(* IEC 61131-3 sources: LTL-Test-Case-Generation/ (part 3) *)

(* ---- SF_ModeSelector_Test.st ---- *)
FUNCTION_BLOCK SF_ModeSelector_Test
VAR_INPUT
END_VAR
VAR_OUTPUT
	failed_0: BOOL := FALSE;
	finished_0: BOOL := FALSE;
END_VAR
VAR
	fb_0: SF_ModeSelector_BranchCounters;
	waitCounter_0: UINT := 0;
	testState_0: UINT := 0;
END_VAR

IF NOT failed_0 AND NOT finished_0 THEN
CASE testState_0 OF
0:
	fb_0.Activate := FALSE;
	fb_0();
	failed_0 := NOT (((((((((((((((((NOT (fb_0.Reset_Before) AND NOT (fb_0.S_SetMode_Before)) AND NOT (fb_0.T_1.Q)) AND (fb_0.DiagCode = 0)) AND NOT (fb_0.Ready)) AND NOT (fb_0.SafetyDemand)) AND NOT (fb_0.ResetRequest)) AND NOT (fb_0.Error)) AND NOT (fb_0.S_AnyModeSel)) AND NOT (fb_0.S_Mode0Sel)) AND NOT (fb_0.S_Mode1Sel)) AND NOT (fb_0.S_Mode2Sel)) AND NOT (fb_0.S_Mode3Sel)) AND NOT (fb_0.S_Mode4Sel)) AND NOT (fb_0.S_Mode5Sel)) AND NOT (fb_0.S_Mode6Sel)) AND NOT (fb_0.S_Mode7Sel)));
	testState_0 := testState_0 + 1;
1:
	fb_0.Activate := TRUE; fb_0.AutoSetMode := TRUE; fb_0.S_SetMode := FALSE; fb_0.S_Unlock := FALSE; fb_0.Reset := FALSE; fb_0.S_Mode0 := FALSE; fb_0.S_Mode1 := FALSE; fb_0.S_Mode2 := FALSE; fb_0.S_Mode3 := FALSE; fb_0.S_Mode4 := FALSE; fb_0.S_Mode5 := FALSE; fb_0.S_Mode6 := FALSE; fb_0.S_Mode7 := FALSE;
	fb_0();
	failed_0 := NOT (((((((((((((((((NOT (fb_0.Reset_Before) AND NOT (fb_0.S_SetMode_Before)) AND NOT (fb_0.T_1.Q)) AND (fb_0.DiagCode = 34818)) AND fb_0.Ready) AND fb_0.SafetyDemand) AND NOT (fb_0.ResetRequest)) AND NOT (fb_0.Error)) AND NOT (fb_0.S_AnyModeSel)) AND NOT (fb_0.S_Mode0Sel)) AND NOT (fb_0.S_Mode1Sel)) AND NOT (fb_0.S_Mode2Sel)) AND NOT (fb_0.S_Mode3Sel)) AND NOT (fb_0.S_Mode4Sel)) AND NOT (fb_0.S_Mode5Sel)) AND NOT (fb_0.S_Mode6Sel)) AND NOT (fb_0.S_Mode7Sel)));
	testState_0 := testState_0 + 1;
2:
	IF fb_0.T_1.Q THEN
		waitCounter_0 := 0;
		testState_0 := testState_0 + 1;
	ELSE
		failed_0 := NOT ((NOT (fb_0.Reset_Before) AND (NOT (fb_0.S_SetMode_Before) AND (NOT (fb_0.T_1.Q) AND ((fb_0.DiagCode = 34818) AND (fb_0.Ready AND (fb_0.SafetyDemand AND (NOT (fb_0.ResetRequest) AND (NOT (fb_0.Error) AND (NOT (fb_0.S_AnyModeSel) AND (NOT (fb_0.S_Mode0Sel) AND (NOT (fb_0.S_Mode1Sel) AND (NOT (fb_0.S_Mode2Sel) AND (NOT (fb_0.S_Mode3Sel) AND (NOT (fb_0.S_Mode4Sel) AND (NOT (fb_0.S_Mode5Sel) AND (NOT (fb_0.S_Mode6Sel) AND NOT (fb_0.S_Mode7Sel))))))))))))))))));
		IF waitCounter_0 > 100 THEN
			finished_0 := TRUE;
		ELSE
			waitCounter_0 := waitCounter_0 + 1;
			fb_0();
		END_IF
	END_IF
3:
	failed_0 := NOT (((((((((((((((((NOT (fb_0.Reset_Before) AND NOT (fb_0.S_SetMode_Before)) AND fb_0.T_1.Q) AND (fb_0.DiagCode = 49184)) AND fb_0.Ready) AND NOT (fb_0.SafetyDemand)) AND NOT (fb_0.ResetRequest)) AND fb_0.Error) AND NOT (fb_0.S_AnyModeSel)) AND NOT (fb_0.S_Mode0Sel)) AND NOT (fb_0.S_Mode1Sel)) AND NOT (fb_0.S_Mode2Sel)) AND NOT (fb_0.S_Mode3Sel)) AND NOT (fb_0.S_Mode4Sel)) AND NOT (fb_0.S_Mode5Sel)) AND NOT (fb_0.S_Mode6Sel)) AND NOT (fb_0.S_Mode7Sel)));
	testState_0 := testState_0 + 1;
4:
	fb_0.Activate := TRUE; fb_0.AutoSetMode := TRUE; fb_0.S_SetMode := FALSE; fb_0.S_Unlock := FALSE; fb_0.Reset := TRUE; fb_0.S_Mode0 := FALSE; fb_0.S_Mode1 := FALSE; fb_0.S_Mode2 := FALSE; fb_0.S_Mode3 := FALSE; fb_0.S_Mode4 := FALSE; fb_0.S_Mode5 := FALSE; fb_0.S_Mode6 := FALSE; fb_0.S_Mode7 := FALSE;
	fb_0();
	failed_0 := NOT (((((((((((((((((fb_0.Reset_Before AND NOT (fb_0.S_SetMode_Before)) AND fb_0.T_1.Q) AND (fb_0.DiagCode = 49184)) AND fb_0.Ready) AND NOT (fb_0.SafetyDemand)) AND NOT (fb_0.ResetRequest)) AND fb_0.Error) AND NOT (fb_0.S_AnyModeSel)) AND NOT (fb_0.S_Mode0Sel)) AND NOT (fb_0.S_Mode1Sel)) AND NOT (fb_0.S_Mode2Sel)) AND NOT (fb_0.S_Mode3Sel)) AND NOT (fb_0.S_Mode4Sel)) AND NOT (fb_0.S_Mode5Sel)) AND NOT (fb_0.S_Mode6Sel)) AND NOT (fb_0.S_Mode7Sel)));
	testState_0 := testState_0 + 1;
5:
	fb_0.Activate := TRUE; fb_0.AutoSetMode := TRUE; fb_0.S_SetMode := FALSE; fb_0.S_Unlock := FALSE; fb_0.Reset := TRUE; fb_0.S_Mode0 := FALSE; fb_0.S_Mode1 := FALSE; fb_0.S_Mode2 := FALSE; fb_0.S_Mode3 := FALSE; fb_0.S_Mode4 := FALSE; fb_0.S_Mode5 := FALSE; fb_0.S_Mode6 := FALSE; fb_0.S_Mode7 := FALSE;
	fb_0();
	failed_0 := NOT (((((((((((((((((fb_0.Reset_Before AND NOT (fb_0.S_SetMode_Before)) AND fb_0.T_1.Q) AND (fb_0.DiagCode = 49185)) AND fb_0.Ready) AND NOT (fb_0.SafetyDemand)) AND NOT (fb_0.ResetRequest)) AND fb_0.Error) AND NOT (fb_0.S_AnyModeSel)) AND NOT (fb_0.S_Mode0Sel)) AND NOT (fb_0.S_Mode1Sel)) AND NOT (fb_0.S_Mode2Sel)) AND NOT (fb_0.S_Mode3Sel)) AND NOT (fb_0.S_Mode4Sel)) AND NOT (fb_0.S_Mode5Sel)) AND NOT (fb_0.S_Mode6Sel)) AND NOT (fb_0.S_Mode7Sel)));
	testState_0 := testState_0 + 1;
6:
	fb_0.Activate := TRUE; fb_0.AutoSetMode := TRUE; fb_0.S_SetMode := FALSE; fb_0.S_Unlock := FALSE; fb_0.Reset := TRUE; fb_0.S_Mode0 := FALSE; fb_0.S_Mode1 := FALSE; fb_0.S_Mode2 := FALSE; fb_0.S_Mode3 := FALSE; fb_0.S_Mode4 := FALSE; fb_0.S_Mode5 := FALSE; fb_0.S_Mode6 := FALSE; fb_0.S_Mode7 := FALSE;
	fb_0();
	failed_0 := NOT (((((((((((((((((fb_0.Reset_Before AND NOT (fb_0.S_SetMode_Before)) AND fb_0.T_1.Q) AND (fb_0.DiagCode = 49185)) AND fb_0.Ready) AND NOT (fb_0.SafetyDemand)) AND NOT (fb_0.ResetRequest)) AND fb_0.Error) AND NOT (fb_0.S_AnyModeSel)) AND NOT (fb_0.S_Mode0Sel)) AND NOT (fb_0.S_Mode1Sel)) AND NOT (fb_0.S_Mode2Sel)) AND NOT (fb_0.S_Mode3Sel)) AND NOT (fb_0.S_Mode4Sel)) AND NOT (fb_0.S_Mode5Sel)) AND NOT (fb_0.S_Mode6Sel)) AND NOT (fb_0.S_Mode7Sel)));
	testState_0 := testState_0 + 1;
7:
	fb_0.Activate := TRUE; fb_0.AutoSetMode := TRUE; fb_0.S_SetMode := FALSE; fb_0.S_Unlock := FALSE; fb_0.Reset := FALSE; fb_0.S_Mode0 := FALSE; fb_0.S_Mode1 := FALSE; fb_0.S_Mode2 := FALSE; fb_0.S_Mode3 := FALSE; fb_0.S_Mode4 := FALSE; fb_0.S_Mode5 := FALSE; fb_0.S_Mode6 := FALSE; fb_0.S_Mode7 := FALSE;
	fb_0();
	failed_0 := NOT (((((((((((((((((NOT (fb_0.Reset_Before) AND NOT (fb_0.S_SetMode_Before)) AND fb_0.T_1.Q) AND (fb_0.DiagCode = 49184)) AND fb_0.Ready) AND NOT (fb_0.SafetyDemand)) AND NOT (fb_0.ResetRequest)) AND fb_0.Error) AND NOT (fb_0.S_AnyModeSel)) AND NOT (fb_0.S_Mode0Sel)) AND NOT (fb_0.S_Mode1Sel)) AND NOT (fb_0.S_Mode2Sel)) AND NOT (fb_0.S_Mode3Sel)) AND NOT (fb_0.S_Mode4Sel)) AND NOT (fb_0.S_Mode5Sel)) AND NOT (fb_0.S_Mode6Sel)) AND NOT (fb_0.S_Mode7Sel)));
	testState_0 := testState_0 + 1;
8:
	fb_0.Activate := TRUE; fb_0.AutoSetMode := TRUE; fb_0.S_SetMode := FALSE; fb_0.S_Unlock := FALSE; fb_0.Reset := FALSE; fb_0.S_Mode0 := FALSE; fb_0.S_Mode1 := TRUE; fb_0.S_Mode2 := FALSE; fb_0.S_Mode3 := FALSE; fb_0.S_Mode4 := FALSE; fb_0.S_Mode5 := FALSE; fb_0.S_Mode6 := FALSE; fb_0.S_Mode7 := FALSE;
	fb_0();
	failed_0 := NOT (((((((((((((((((NOT (fb_0.Reset_Before) AND NOT (fb_0.S_SetMode_Before)) AND fb_0.T_1.Q) AND (fb_0.DiagCode = 50208)) AND fb_0.Ready) AND NOT (fb_0.SafetyDemand)) AND fb_0.ResetRequest) AND fb_0.Error) AND NOT (fb_0.S_AnyModeSel)) AND NOT (fb_0.S_Mode0Sel)) AND NOT (fb_0.S_Mode1Sel)) AND NOT (fb_0.S_Mode2Sel)) AND NOT (fb_0.S_Mode3Sel)) AND NOT (fb_0.S_Mode4Sel)) AND NOT (fb_0.S_Mode5Sel)) AND NOT (fb_0.S_Mode6Sel)) AND NOT (fb_0.S_Mode7Sel)));
	testState_0 := testState_0 + 1;
9:
	fb_0.Activate := TRUE; fb_0.AutoSetMode := TRUE; fb_0.S_SetMode := FALSE; fb_0.S_Unlock := FALSE; fb_0.Reset := FALSE; fb_0.S_Mode0 := FALSE; fb_0.S_Mode1 := FALSE; fb_0.S_Mode2 := FALSE; fb_0.S_Mode3 := FALSE; fb_0.S_Mode4 := FALSE; fb_0.S_Mode5 := FALSE; fb_0.S_Mode6 := FALSE; fb_0.S_Mode7 := FALSE;
	fb_0();
	failed_0 := NOT (((((((((((((((((NOT (fb_0.Reset_Before) AND NOT (fb_0.S_SetMode_Before)) AND fb_0.T_1.Q) AND (fb_0.DiagCode = 49184)) AND fb_0.Ready) AND NOT (fb_0.SafetyDemand)) AND NOT (fb_0.ResetRequest)) AND fb_0.Error) AND NOT (fb_0.S_AnyModeSel)) AND NOT (fb_0.S_Mode0Sel)) AND NOT (fb_0.S_Mode1Sel)) AND NOT (fb_0.S_Mode2Sel)) AND NOT (fb_0.S_Mode3Sel)) AND NOT (fb_0.S_Mode4Sel)) AND NOT (fb_0.S_Mode5Sel)) AND NOT (fb_0.S_Mode6Sel)) AND NOT (fb_0.S_Mode7Sel)));
	testState_0 := testState_0 + 1;
10:
	fb_0.Activate := TRUE; fb_0.AutoSetMode := TRUE; fb_0.S_SetMode := FALSE; fb_0.S_Unlock := FALSE; fb_0.Reset := FALSE; fb_0.S_Mode0 := FALSE; fb_0.S_Mode1 := TRUE; fb_0.S_Mode2 := FALSE; fb_0.S_Mode3 := FALSE; fb_0.S_Mode4 := FALSE; fb_0.S_Mode5 := FALSE; fb_0.S_Mode6 := FALSE; fb_0.S_Mode7 := FALSE;
	fb_0();
	failed_0 := NOT (((((((((((((((((NOT (fb_0.Reset_Before) AND NOT (fb_0.S_SetMode_Before)) AND fb_0.T_1.Q) AND (fb_0.DiagCode = 50208)) AND fb_0.Ready) AND NOT (fb_0.SafetyDemand)) AND fb_0.ResetRequest) AND fb_0.Error) AND NOT (fb_0.S_AnyModeSel)) AND NOT (fb_0.S_Mode0Sel)) AND NOT (fb_0.S_Mode1Sel)) AND NOT (fb_0.S_Mode2Sel)) AND NOT (fb_0.S_Mode3Sel)) AND NOT (fb_0.S_Mode4Sel)) AND NOT (fb_0.S_Mode5Sel)) AND NOT (fb_0.S_Mode6Sel)) AND NOT (fb_0.S_Mode7Sel)));
	testState_0 := testState_0 + 1;
11:
	fb_0.Activate := TRUE; fb_0.AutoSetMode := TRUE; fb_0.S_SetMode := FALSE; fb_0.S_Unlock := FALSE; fb_0.Reset := FALSE; fb_0.S_Mode0 := FALSE; fb_0.S_Mode1 := TRUE; fb_0.S_Mode2 := FALSE; fb_0.S_Mode3 := FALSE; fb_0.S_Mode4 := FALSE; fb_0.S_Mode5 := FALSE; fb_0.S_Mode6 := FALSE; fb_0.S_Mode7 := FALSE;
	fb_0();
	failed_0 := NOT (((((((((((((((((NOT (fb_0.Reset_Before) AND NOT (fb_0.S_SetMode_Before)) AND fb_0.T_1.Q) AND (fb_0.DiagCode = 50208)) AND fb_0.Ready) AND NOT (fb_0.SafetyDemand)) AND fb_0.ResetRequest) AND fb_0.Error) AND NOT (fb_0.S_AnyModeSel)) AND NOT (fb_0.S_Mode0Sel)) AND NOT (fb_0.S_Mode1Sel)) AND NOT (fb_0.S_Mode2Sel)) AND NOT (fb_0.S_Mode3Sel)) AND NOT (fb_0.S_Mode4Sel)) AND NOT (fb_0.S_Mode5Sel)) AND NOT (fb_0.S_Mode6Sel)) AND NOT (fb_0.S_Mode7Sel)));
	testState_0 := testState_0 + 1;
12:
	fb_0.Activate := TRUE; fb_0.AutoSetMode := TRUE; fb_0.S_SetMode := FALSE; fb_0.S_Unlock := FALSE; fb_0.Reset := TRUE; fb_0.S_Mode0 := FALSE; fb_0.S_Mode1 := TRUE; fb_0.S_Mode2 := FALSE; fb_0.S_Mode3 := FALSE; fb_0.S_Mode4 := FALSE; fb_0.S_Mode5 := FALSE; fb_0.S_Mode6 := FALSE; fb_0.S_Mode7 := FALSE;
	fb_0();
	failed_0 := NOT (((((((((((((((((fb_0.Reset_Before AND NOT (fb_0.S_SetMode_Before)) AND NOT (fb_0.T_1.Q)) AND (fb_0.DiagCode = 34818)) AND fb_0.Ready) AND fb_0.SafetyDemand) AND NOT (fb_0.ResetRequest)) AND NOT (fb_0.Error)) AND NOT (fb_0.S_AnyModeSel)) AND NOT (fb_0.S_Mode0Sel)) AND NOT (fb_0.S_Mode1Sel)) AND NOT (fb_0.S_Mode2Sel)) AND NOT (fb_0.S_Mode3Sel)) AND NOT (fb_0.S_Mode4Sel)) AND NOT (fb_0.S_Mode5Sel)) AND NOT (fb_0.S_Mode6Sel)) AND NOT (fb_0.S_Mode7Sel)));
	testState_0 := testState_0 + 1;
13:
	fb_0.Activate := TRUE; fb_0.AutoSetMode := TRUE; fb_0.S_SetMode := FALSE; fb_0.S_Unlock := FALSE; fb_0.Reset := FALSE; fb_0.S_Mode0 := FALSE; fb_0.S_Mode1 := FALSE; fb_0.S_Mode2 := FALSE; fb_0.S_Mode3 := FALSE; fb_0.S_Mode4 := FALSE; fb_0.S_Mode5 := FALSE; fb_0.S_Mode6 := FALSE; fb_0.S_Mode7 := FALSE;
	fb_0();
	failed_0 := NOT (((((((((((((((((NOT (fb_0.Reset_Before) AND NOT (fb_0.S_SetMode_Before)) AND NOT (fb_0.T_1.Q)) AND (fb_0.DiagCode = 34818)) AND fb_0.Ready) AND fb_0.SafetyDemand) AND NOT (fb_0.ResetRequest)) AND NOT (fb_0.Error)) AND NOT (fb_0.S_AnyModeSel)) AND NOT (fb_0.S_Mode0Sel)) AND NOT (fb_0.S_Mode1Sel)) AND NOT (fb_0.S_Mode2Sel)) AND NOT (fb_0.S_Mode3Sel)) AND NOT (fb_0.S_Mode4Sel)) AND NOT (fb_0.S_Mode5Sel)) AND NOT (fb_0.S_Mode6Sel)) AND NOT (fb_0.S_Mode7Sel)));
	testState_0 := testState_0 + 1;
14:
	IF fb_0.T_1.Q THEN
		waitCounter_0 := 0;
		testState_0 := testState_0 + 1;
	ELSE
		failed_0 := NOT ((NOT (fb_0.Reset_Before) AND (NOT (fb_0.S_SetMode_Before) AND (NOT (fb_0.T_1.Q) AND ((fb_0.DiagCode = 34818) AND (fb_0.Ready AND (fb_0.SafetyDemand AND (NOT (fb_0.ResetRequest) AND (NOT (fb_0.Error) AND (NOT (fb_0.S_AnyModeSel) AND (NOT (fb_0.S_Mode0Sel) AND (NOT (fb_0.S_Mode1Sel) AND (NOT (fb_0.S_Mode2Sel) AND (NOT (fb_0.S_Mode3Sel) AND (NOT (fb_0.S_Mode4Sel) AND (NOT (fb_0.S_Mode5Sel) AND (NOT (fb_0.S_Mode6Sel) AND NOT (fb_0.S_Mode7Sel))))))))))))))))));
		IF waitCounter_0 > 100 THEN
			finished_0 := TRUE;
		ELSE
			waitCounter_0 := waitCounter_0 + 1;
			fb_0();
		END_IF
	END_IF
15:
	failed_0 := NOT (((((((((((((((((NOT (fb_0.Reset_Before) AND NOT (fb_0.S_SetMode_Before)) AND fb_0.T_1.Q) AND (fb_0.DiagCode = 49184)) AND fb_0.Ready) AND NOT (fb_0.SafetyDemand)) AND NOT (fb_0.ResetRequest)) AND fb_0.Error) AND NOT (fb_0.S_AnyModeSel)) AND NOT (fb_0.S_Mode0Sel)) AND NOT (fb_0.S_Mode1Sel)) AND NOT (fb_0.S_Mode2Sel)) AND NOT (fb_0.S_Mode3Sel)) AND NOT (fb_0.S_Mode4Sel)) AND NOT (fb_0.S_Mode5Sel)) AND NOT (fb_0.S_Mode6Sel)) AND NOT (fb_0.S_Mode7Sel)));
	testState_0 := testState_0 + 1;
16:
	fb_0.Activate := TRUE; fb_0.AutoSetMode := TRUE; fb_0.S_SetMode := FALSE; fb_0.S_Unlock := FALSE; fb_0.Reset := TRUE; fb_0.S_Mode0 := FALSE; fb_0.S_Mode1 := TRUE; fb_0.S_Mode2 := FALSE; fb_0.S_Mode3 := FALSE; fb_0.S_Mode4 := FALSE; fb_0.S_Mode5 := FALSE; fb_0.S_Mode6 := FALSE; fb_0.S_Mode7 := FALSE;
	fb_0();
	failed_0 := NOT (((((((((((((((((fb_0.Reset_Before AND NOT (fb_0.S_SetMode_Before)) AND NOT (fb_0.T_1.Q)) AND (fb_0.DiagCode = 34818)) AND fb_0.Ready) AND fb_0.SafetyDemand) AND NOT (fb_0.ResetRequest)) AND NOT (fb_0.Error)) AND NOT (fb_0.S_AnyModeSel)) AND NOT (fb_0.S_Mode0Sel)) AND NOT (fb_0.S_Mode1Sel)) AND NOT (fb_0.S_Mode2Sel)) AND NOT (fb_0.S_Mode3Sel)) AND NOT (fb_0.S_Mode4Sel)) AND NOT (fb_0.S_Mode5Sel)) AND NOT (fb_0.S_Mode6Sel)) AND NOT (fb_0.S_Mode7Sel)));
	testState_0 := testState_0 + 1;
17:
	fb_0.Activate := TRUE; fb_0.AutoSetMode := TRUE; fb_0.S_SetMode := FALSE; fb_0.S_Unlock := FALSE; fb_0.Reset := FALSE; fb_0.S_Mode0 := FALSE; fb_0.S_Mode1 := TRUE; fb_0.S_Mode2 := TRUE; fb_0.S_Mode3 := FALSE; fb_0.S_Mode4 := FALSE; fb_0.S_Mode5 := FALSE; fb_0.S_Mode6 := FALSE; fb_0.S_Mode7 := FALSE;
	fb_0();
	failed_0 := NOT (((((((((((((((((NOT (fb_0.Reset_Before) AND NOT (fb_0.S_SetMode_Before)) AND NOT (fb_0.T_1.Q)) AND (fb_0.DiagCode = 49168)) AND fb_0.Ready) AND NOT (fb_0.SafetyDemand)) AND NOT (fb_0.ResetRequest)) AND fb_0.Error) AND NOT (fb_0.S_AnyModeSel)) AND NOT (fb_0.S_Mode0Sel)) AND NOT (fb_0.S_Mode1Sel)) AND NOT (fb_0.S_Mode2Sel)) AND NOT (fb_0.S_Mode3Sel)) AND NOT (fb_0.S_Mode4Sel)) AND NOT (fb_0.S_Mode5Sel)) AND NOT (fb_0.S_Mode6Sel)) AND NOT (fb_0.S_Mode7Sel)));
	testState_0 := testState_0 + 1;
18:
	fb_0.Activate := TRUE; fb_0.AutoSetMode := TRUE; fb_0.S_SetMode := FALSE; fb_0.S_Unlock := FALSE; fb_0.Reset := TRUE; fb_0.S_Mode0 := FALSE; fb_0.S_Mode1 := TRUE; fb_0.S_Mode2 := TRUE; fb_0.S_Mode3 := FALSE; fb_0.S_Mode4 := FALSE; fb_0.S_Mode5 := FALSE; fb_0.S_Mode6 := FALSE; fb_0.S_Mode7 := FALSE;
	fb_0();
	failed_0 := NOT (((((((((((((((((fb_0.Reset_Before AND NOT (fb_0.S_SetMode_Before)) AND NOT (fb_0.T_1.Q)) AND (fb_0.DiagCode = 49168)) AND fb_0.Ready) AND NOT (fb_0.SafetyDemand)) AND NOT (fb_0.ResetRequest)) AND fb_0.Error) AND NOT (fb_0.S_AnyModeSel)) AND NOT (fb_0.S_Mode0Sel)) AND NOT (fb_0.S_Mode1Sel)) AND NOT (fb_0.S_Mode2Sel)) AND NOT (fb_0.S_Mode3Sel)) AND NOT (fb_0.S_Mode4Sel)) AND NOT (fb_0.S_Mode5Sel)) AND NOT (fb_0.S_Mode6Sel)) AND NOT (fb_0.S_Mode7Sel)));
	testState_0 := testState_0 + 1;
19:
	fb_0.Activate := TRUE; fb_0.AutoSetMode := TRUE; fb_0.S_SetMode := FALSE; fb_0.S_Unlock := FALSE; fb_0.Reset := TRUE; fb_0.S_Mode0 := FALSE; fb_0.S_Mode1 := TRUE; fb_0.S_Mode2 := TRUE; fb_0.S_Mode3 := FALSE; fb_0.S_Mode4 := FALSE; fb_0.S_Mode5 := FALSE; fb_0.S_Mode6 := FALSE; fb_0.S_Mode7 := FALSE;
	fb_0();
	failed_0 := NOT (((((((((((((((((fb_0.Reset_Before AND NOT (fb_0.S_SetMode_Before)) AND NOT (fb_0.T_1.Q)) AND (fb_0.DiagCode = 49169)) AND fb_0.Ready) AND NOT (fb_0.SafetyDemand)) AND NOT (fb_0.ResetRequest)) AND fb_0.Error) AND NOT (fb_0.S_AnyModeSel)) AND NOT (fb_0.S_Mode0Sel)) AND NOT (fb_0.S_Mode1Sel)) AND NOT (fb_0.S_Mode2Sel)) AND NOT (fb_0.S_Mode3Sel)) AND NOT (fb_0.S_Mode4Sel)) AND NOT (fb_0.S_Mode5Sel)) AND NOT (fb_0.S_Mode6Sel)) AND NOT (fb_0.S_Mode7Sel)));
	testState_0 := testState_0 + 1;
20:
	fb_0.Activate := TRUE; fb_0.AutoSetMode := TRUE; fb_0.S_SetMode := FALSE; fb_0.S_Unlock := FALSE; fb_0.Reset := TRUE; fb_0.S_Mode0 := FALSE; fb_0.S_Mode1 := TRUE; fb_0.S_Mode2 := TRUE; fb_0.S_Mode3 := FALSE; fb_0.S_Mode4 := FALSE; fb_0.S_Mode5 := FALSE; fb_0.S_Mode6 := FALSE; fb_0.S_Mode7 := FALSE;
	fb_0();
	failed_0 := NOT (((((((((((((((((fb_0.Reset_Before AND NOT (fb_0.S_SetMode_Before)) AND NOT (fb_0.T_1.Q)) AND (fb_0.DiagCode = 49169)) AND fb_0.Ready) AND NOT (fb_0.SafetyDemand)) AND NOT (fb_0.ResetRequest)) AND fb_0.Error) AND NOT (fb_0.S_AnyModeSel)) AND NOT (fb_0.S_Mode0Sel)) AND NOT (fb_0.S_Mode1Sel)) AND NOT (fb_0.S_Mode2Sel)) AND NOT (fb_0.S_Mode3Sel)) AND NOT (fb_0.S_Mode4Sel)) AND NOT (fb_0.S_Mode5Sel)) AND NOT (fb_0.S_Mode6Sel)) AND NOT (fb_0.S_Mode7Sel)));
	testState_0 := testState_0 + 1;
21:
	fb_0.Activate := TRUE; fb_0.AutoSetMode := TRUE; fb_0.S_SetMode := FALSE; fb_0.S_Unlock := FALSE; fb_0.Reset := FALSE; fb_0.S_Mode0 := FALSE; fb_0.S_Mode1 := TRUE; fb_0.S_Mode2 := TRUE; fb_0.S_Mode3 := FALSE; fb_0.S_Mode4 := FALSE; fb_0.S_Mode5 := FALSE; fb_0.S_Mode6 := FALSE; fb_0.S_Mode7 := FALSE;
	fb_0();
	failed_0 := NOT (((((((((((((((((NOT (fb_0.Reset_Before) AND NOT (fb_0.S_SetMode_Before)) AND NOT (fb_0.T_1.Q)) AND (fb_0.DiagCode = 49168)) AND fb_0.Ready) AND NOT (fb_0.SafetyDemand)) AND NOT (fb_0.ResetRequest)) AND fb_0.Error) AND NOT (fb_0.S_AnyModeSel)) AND NOT (fb_0.S_Mode0Sel)) AND NOT (fb_0.S_Mode1Sel)) AND NOT (fb_0.S_Mode2Sel)) AND NOT (fb_0.S_Mode3Sel)) AND NOT (fb_0.S_Mode4Sel)) AND NOT (fb_0.S_Mode5Sel)) AND NOT (fb_0.S_Mode6Sel)) AND NOT (fb_0.S_Mode7Sel)));
	testState_0 := testState_0 + 1;
22:
	fb_0.Activate := TRUE; fb_0.AutoSetMode := TRUE; fb_0.S_SetMode := FALSE; fb_0.S_Unlock := FALSE; fb_0.Reset := FALSE; fb_0.S_Mode0 := FALSE; fb_0.S_Mode1 := FALSE; fb_0.S_Mode2 := FALSE; fb_0.S_Mode3 := FALSE; fb_0.S_Mode4 := FALSE; fb_0.S_Mode5 := FALSE; fb_0.S_Mode6 := FALSE; fb_0.S_Mode7 := FALSE;
	fb_0();
	failed_0 := NOT (((((((((((((((((NOT (fb_0.Reset_Before) AND NOT (fb_0.S_SetMode_Before)) AND NOT (fb_0.T_1.Q)) AND (fb_0.DiagCode = 50192)) AND fb_0.Ready) AND NOT (fb_0.SafetyDemand)) AND fb_0.ResetRequest) AND fb_0.Error) AND NOT (fb_0.S_AnyModeSel)) AND NOT (fb_0.S_Mode0Sel)) AND NOT (fb_0.S_Mode1Sel)) AND NOT (fb_0.S_Mode2Sel)) AND NOT (fb_0.S_Mode3Sel)) AND NOT (fb_0.S_Mode4Sel)) AND NOT (fb_0.S_Mode5Sel)) AND NOT (fb_0.S_Mode6Sel)) AND NOT (fb_0.S_Mode7Sel)));
	testState_0 := testState_0 + 1;
23:
	fb_0.Activate := TRUE; fb_0.AutoSetMode := TRUE; fb_0.S_SetMode := FALSE; fb_0.S_Unlock := FALSE; fb_0.Reset := FALSE; fb_0.S_Mode0 := FALSE; fb_0.S_Mode1 := TRUE; fb_0.S_Mode2 := TRUE; fb_0.S_Mode3 := FALSE; fb_0.S_Mode4 := FALSE; fb_0.S_Mode5 := FALSE; fb_0.S_Mode6 := FALSE; fb_0.S_Mode7 := FALSE;
	fb_0();
	failed_0 := NOT (((((((((((((((((NOT (fb_0.Reset_Before) AND NOT (fb_0.S_SetMode_Before)) AND NOT (fb_0.T_1.Q)) AND (fb_0.DiagCode = 49168)) AND fb_0.Ready) AND NOT (fb_0.SafetyDemand)) AND NOT (fb_0.ResetRequest)) AND fb_0.Error) AND NOT (fb_0.S_AnyModeSel)) AND NOT (fb_0.S_Mode0Sel)) AND NOT (fb_0.S_Mode1Sel)) AND NOT (fb_0.S_Mode2Sel)) AND NOT (fb_0.S_Mode3Sel)) AND NOT (fb_0.S_Mode4Sel)) AND NOT (fb_0.S_Mode5Sel)) AND NOT (fb_0.S_Mode6Sel)) AND NOT (fb_0.S_Mode7Sel)));
	testState_0 := testState_0 + 1;
24:
	fb_0.Activate := TRUE; fb_0.AutoSetMode := TRUE; fb_0.S_SetMode := FALSE; fb_0.S_Unlock := FALSE; fb_0.Reset := FALSE; fb_0.S_Mode0 := FALSE; fb_0.S_Mode1 := FALSE; fb_0.S_Mode2 := FALSE; fb_0.S_Mode3 := FALSE; fb_0.S_Mode4 := FALSE; fb_0.S_Mode5 := FALSE; fb_0.S_Mode6 := FALSE; fb_0.S_Mode7 := FALSE;
	fb_0();
	failed_0 := NOT (((((((((((((((((NOT (fb_0.Reset_Before) AND NOT (fb_0.S_SetMode_Before)) AND NOT (fb_0.T_1.Q)) AND (fb_0.DiagCode = 50192)) AND fb_0.Ready) AND NOT (fb_0.SafetyDemand)) AND fb_0.ResetRequest) AND fb_0.Error) AND NOT (fb_0.S_AnyModeSel)) AND NOT (fb_0.S_Mode0Sel)) AND NOT (fb_0.S_Mode1Sel)) AND NOT (fb_0.S_Mode2Sel)) AND NOT (fb_0.S_Mode3Sel)) AND NOT (fb_0.S_Mode4Sel)) AND NOT (fb_0.S_Mode5Sel)) AND NOT (fb_0.S_Mode6Sel)) AND NOT (fb_0.S_Mode7Sel)));
	testState_0 := testState_0 + 1;
25:
	fb_0.Activate := TRUE; fb_0.AutoSetMode := TRUE; fb_0.S_SetMode := FALSE; fb_0.S_Unlock := FALSE; fb_0.Reset := FALSE; fb_0.S_Mode0 := FALSE; fb_0.S_Mode1 := FALSE; fb_0.S_Mode2 := FALSE; fb_0.S_Mode3 := FALSE; fb_0.S_Mode4 := FALSE; fb_0.S_Mode5 := FALSE; fb_0.S_Mode6 := FALSE; fb_0.S_Mode7 := FALSE;
	fb_0();
	failed_0 := NOT (((((((((((((((((NOT (fb_0.Reset_Before) AND NOT (fb_0.S_SetMode_Before)) AND NOT (fb_0.T_1.Q)) AND (fb_0.DiagCode = 50192)) AND fb_0.Ready) AND NOT (fb_0.SafetyDemand)) AND fb_0.ResetRequest) AND fb_0.Error) AND NOT (fb_0.S_AnyModeSel)) AND NOT (fb_0.S_Mode0Sel)) AND NOT (fb_0.S_Mode1Sel)) AND NOT (fb_0.S_Mode2Sel)) AND NOT (fb_0.S_Mode3Sel)) AND NOT (fb_0.S_Mode4Sel)) AND NOT (fb_0.S_Mode5Sel)) AND NOT (fb_0.S_Mode6Sel)) AND NOT (fb_0.S_Mode7Sel)));
	testState_0 := testState_0 + 1;
26:
	fb_0.Activate := TRUE; fb_0.AutoSetMode := TRUE; fb_0.S_SetMode := FALSE; fb_0.S_Unlock := FALSE; fb_0.Reset := TRUE; fb_0.S_Mode0 := FALSE; fb_0.S_Mode1 := FALSE; fb_0.S_Mode2 := FALSE; fb_0.S_Mode3 := FALSE; fb_0.S_Mode4 := FALSE; fb_0.S_Mode5 := FALSE; fb_0.S_Mode6 := FALSE; fb_0.S_Mode7 := FALSE;
	fb_0();
	failed_0 := NOT (((((((((((((((((fb_0.Reset_Before AND NOT (fb_0.S_SetMode_Before)) AND NOT (fb_0.T_1.Q)) AND (fb_0.DiagCode = 34818)) AND fb_0.Ready) AND fb_0.SafetyDemand) AND NOT (fb_0.ResetRequest)) AND NOT (fb_0.Error)) AND NOT (fb_0.S_AnyModeSel)) AND NOT (fb_0.S_Mode0Sel)) AND NOT (fb_0.S_Mode1Sel)) AND NOT (fb_0.S_Mode2Sel)) AND NOT (fb_0.S_Mode3Sel)) AND NOT (fb_0.S_Mode4Sel)) AND NOT (fb_0.S_Mode5Sel)) AND NOT (fb_0.S_Mode6Sel)) AND NOT (fb_0.S_Mode7Sel)));
	testState_0 := testState_0 + 1;
27:
	fb_0.Activate := TRUE; fb_0.AutoSetMode := TRUE; fb_0.S_SetMode := FALSE; fb_0.S_Unlock := FALSE; fb_0.Reset := FALSE; fb_0.S_Mode0 := FALSE; fb_0.S_Mode1 := FALSE; fb_0.S_Mode2 := TRUE; fb_0.S_Mode3 := TRUE; fb_0.S_Mode4 := FALSE; fb_0.S_Mode5 := FALSE; fb_0.S_Mode6 := FALSE; fb_0.S_Mode7 := FALSE;
	fb_0();
	failed_0 := NOT (((((((((((((((((NOT (fb_0.Reset_Before) AND NOT (fb_0.S_SetMode_Before)) AND NOT (fb_0.T_1.Q)) AND (fb_0.DiagCode = 49168)) AND fb_0.Ready) AND NOT (fb_0.SafetyDemand)) AND NOT (fb_0.ResetRequest)) AND fb_0.Error) AND NOT (fb_0.S_AnyModeSel)) AND NOT (fb_0.S_Mode0Sel)) AND NOT (fb_0.S_Mode1Sel)) AND NOT (fb_0.S_Mode2Sel)) AND NOT (fb_0.S_Mode3Sel)) AND NOT (fb_0.S_Mode4Sel)) AND NOT (fb_0.S_Mode5Sel)) AND NOT (fb_0.S_Mode6Sel)) AND NOT (fb_0.S_Mode7Sel)));
	testState_0 := testState_0 + 1;
28:
	fb_0.Activate := TRUE; fb_0.AutoSetMode := TRUE; fb_0.S_SetMode := FALSE; fb_0.S_Unlock := FALSE; fb_0.Reset := TRUE; fb_0.S_Mode0 := FALSE; fb_0.S_Mode1 := FALSE; fb_0.S_Mode2 := FALSE; fb_0.S_Mode3 := FALSE; fb_0.S_Mode4 := FALSE; fb_0.S_Mode5 := FALSE; fb_0.S_Mode6 := FALSE; fb_0.S_Mode7 := FALSE;
	fb_0();
	failed_0 := NOT (((((((((((((((((fb_0.Reset_Before AND NOT (fb_0.S_SetMode_Before)) AND NOT (fb_0.T_1.Q)) AND (fb_0.DiagCode = 34818)) AND fb_0.Ready) AND fb_0.SafetyDemand) AND NOT (fb_0.ResetRequest)) AND NOT (fb_0.Error)) AND NOT (fb_0.S_AnyModeSel)) AND NOT (fb_0.S_Mode0Sel)) AND NOT (fb_0.S_Mode1Sel)) AND NOT (fb_0.S_Mode2Sel)) AND NOT (fb_0.S_Mode3Sel)) AND NOT (fb_0.S_Mode4Sel)) AND NOT (fb_0.S_Mode5Sel)) AND NOT (fb_0.S_Mode6Sel)) AND NOT (fb_0.S_Mode7Sel)));
	testState_0 := testState_0 + 1;
29:
	fb_0.Activate := TRUE; fb_0.AutoSetMode := TRUE; fb_0.S_SetMode := FALSE; fb_0.S_Unlock := FALSE; fb_0.Reset := FALSE; fb_0.S_Mode0 := FALSE; fb_0.S_Mode1 := FALSE; fb_0.S_Mode2 := FALSE; fb_0.S_Mode3 := FALSE; fb_0.S_Mode4 := FALSE; fb_0.S_Mode5 := FALSE; fb_0.S_Mode6 := FALSE; fb_0.S_Mode7 := FALSE;
	fb_0();
	failed_0 := NOT (((((((((((((((((NOT (fb_0.Reset_Before) AND NOT (fb_0.S_SetMode_Before)) AND NOT (fb_0.T_1.Q)) AND (fb_0.DiagCode = 34818)) AND fb_0.Ready) AND fb_0.SafetyDemand) AND NOT (fb_0.ResetRequest)) AND NOT (fb_0.Error)) AND NOT (fb_0.S_AnyModeSel)) AND NOT (fb_0.S_Mode0Sel)) AND NOT (fb_0.S_Mode1Sel)) AND NOT (fb_0.S_Mode2Sel)) AND NOT (fb_0.S_Mode3Sel)) AND NOT (fb_0.S_Mode4Sel)) AND NOT (fb_0.S_Mode5Sel)) AND NOT (fb_0.S_Mode6Sel)) AND NOT (fb_0.S_Mode7Sel)));
	testState_0 := testState_0 + 1;
30:
	fb_0.Activate := TRUE; fb_0.AutoSetMode := TRUE; fb_0.S_SetMode := FALSE; fb_0.S_Unlock := TRUE; fb_0.Reset := FALSE; fb_0.S_Mode0 := TRUE; fb_0.S_Mode1 := FALSE; fb_0.S_Mode2 := FALSE; fb_0.S_Mode3 := FALSE; fb_0.S_Mode4 := FALSE; fb_0.S_Mode5 := FALSE; fb_0.S_Mode6 := FALSE; fb_0.S_Mode7 := FALSE;
	fb_0();
	failed_0 := NOT (((((((((((((((((NOT (fb_0.Reset_Before) AND NOT (fb_0.S_SetMode_Before)) AND NOT (fb_0.T_1.Q)) AND (fb_0.DiagCode = 32768)) AND fb_0.Ready) AND NOT (fb_0.SafetyDemand)) AND NOT (fb_0.ResetRequest)) AND NOT (fb_0.Error)) AND fb_0.S_AnyModeSel) AND fb_0.S_Mode0Sel) AND NOT (fb_0.S_Mode1Sel)) AND NOT (fb_0.S_Mode2Sel)) AND NOT (fb_0.S_Mode3Sel)) AND NOT (fb_0.S_Mode4Sel)) AND NOT (fb_0.S_Mode5Sel)) AND NOT (fb_0.S_Mode6Sel)) AND NOT (fb_0.S_Mode7Sel)));
	testState_0 := testState_0 + 1;
31:
	fb_0.Activate := TRUE; fb_0.AutoSetMode := TRUE; fb_0.S_SetMode := FALSE; fb_0.S_Unlock := FALSE; fb_0.Reset := FALSE; fb_0.S_Mode0 := TRUE; fb_0.S_Mode1 := FALSE; fb_0.S_Mode2 := FALSE; fb_0.S_Mode3 := FALSE; fb_0.S_Mode4 := FALSE; fb_0.S_Mode5 := FALSE; fb_0.S_Mode6 := FALSE; fb_0.S_Mode7 := FALSE;
	fb_0();
	failed_0 := NOT (((((((((((((((((NOT (fb_0.Reset_Before) AND NOT (fb_0.S_SetMode_Before)) AND NOT (fb_0.T_1.Q)) AND (fb_0.DiagCode = 32784)) AND fb_0.Ready) AND NOT (fb_0.SafetyDemand)) AND NOT (fb_0.ResetRequest)) AND NOT (fb_0.Error)) AND fb_0.S_AnyModeSel) AND fb_0.S_Mode0Sel) AND NOT (fb_0.S_Mode1Sel)) AND NOT (fb_0.S_Mode2Sel)) AND NOT (fb_0.S_Mode3Sel)) AND NOT (fb_0.S_Mode4Sel)) AND NOT (fb_0.S_Mode5Sel)) AND NOT (fb_0.S_Mode6Sel)) AND NOT (fb_0.S_Mode7Sel)));
	testState_0 := testState_0 + 1;
32:
	fb_0.Activate := TRUE; fb_0.AutoSetMode := TRUE; fb_0.S_SetMode := FALSE; fb_0.S_Unlock := TRUE; fb_0.Reset := FALSE; fb_0.S_Mode0 := TRUE; fb_0.S_Mode1 := FALSE; fb_0.S_Mode2 := FALSE; fb_0.S_Mode3 := FALSE; fb_0.S_Mode4 := FALSE; fb_0.S_Mode5 := FALSE; fb_0.S_Mode6 := FALSE; fb_0.S_Mode7 := FALSE;
	fb_0();
	failed_0 := NOT (((((((((((((((((NOT (fb_0.Reset_Before) AND NOT (fb_0.S_SetMode_Before)) AND NOT (fb_0.T_1.Q)) AND (fb_0.DiagCode = 32768)) AND fb_0.Ready) AND NOT (fb_0.SafetyDemand)) AND NOT (fb_0.ResetRequest)) AND NOT (fb_0.Error)) AND fb_0.S_AnyModeSel) AND fb_0.S_Mode0Sel) AND NOT (fb_0.S_Mode1Sel)) AND NOT (fb_0.S_Mode2Sel)) AND NOT (fb_0.S_Mode3Sel)) AND NOT (fb_0.S_Mode4Sel)) AND NOT (fb_0.S_Mode5Sel)) AND NOT (fb_0.S_Mode6Sel)) AND NOT (fb_0.S_Mode7Sel)));
	testState_0 := testState_0 + 1;
33:
	fb_0.Activate := TRUE; fb_0.AutoSetMode := TRUE; fb_0.S_SetMode := FALSE; fb_0.S_Unlock := FALSE; fb_0.Reset := FALSE; fb_0.S_Mode0 := FALSE; fb_0.S_Mode1 := FALSE; fb_0.S_Mode2 := FALSE; fb_0.S_Mode3 := FALSE; fb_0.S_Mode4 := FALSE; fb_0.S_Mode5 := FALSE; fb_0.S_Mode6 := FALSE; fb_0.S_Mode7 := FALSE;
	fb_0();
	failed_0 := NOT (((((((((((((((((NOT (fb_0.Reset_Before) AND NOT (fb_0.S_SetMode_Before)) AND NOT (fb_0.T_1.Q)) AND (fb_0.DiagCode = 34818)) AND fb_0.Ready) AND fb_0.SafetyDemand) AND NOT (fb_0.ResetRequest)) AND NOT (fb_0.Error)) AND NOT (fb_0.S_AnyModeSel)) AND NOT (fb_0.S_Mode0Sel)) AND NOT (fb_0.S_Mode1Sel)) AND NOT (fb_0.S_Mode2Sel)) AND NOT (fb_0.S_Mode3Sel)) AND NOT (fb_0.S_Mode4Sel)) AND NOT (fb_0.S_Mode5Sel)) AND NOT (fb_0.S_Mode6Sel)) AND NOT (fb_0.S_Mode7Sel)));
	testState_0 := testState_0 + 1;
34:
	fb_0.Activate := TRUE; fb_0.AutoSetMode := TRUE; fb_0.S_SetMode := FALSE; fb_0.S_Unlock := TRUE; fb_0.Reset := FALSE; fb_0.S_Mode0 := FALSE; fb_0.S_Mode1 := TRUE; fb_0.S_Mode2 := FALSE; fb_0.S_Mode3 := FALSE; fb_0.S_Mode4 := FALSE; fb_0.S_Mode5 := FALSE; fb_0.S_Mode6 := FALSE; fb_0.S_Mode7 := FALSE;
	fb_0();
	failed_0 := NOT (((((((((((((((((NOT (fb_0.Reset_Before) AND NOT (fb_0.S_SetMode_Before)) AND NOT (fb_0.T_1.Q)) AND (fb_0.DiagCode = 32768)) AND fb_0.Ready) AND NOT (fb_0.SafetyDemand)) AND NOT (fb_0.ResetRequest)) AND NOT (fb_0.Error)) AND fb_0.S_AnyModeSel) AND NOT (fb_0.S_Mode0Sel)) AND fb_0.S_Mode1Sel) AND NOT (fb_0.S_Mode2Sel)) AND NOT (fb_0.S_Mode3Sel)) AND NOT (fb_0.S_Mode4Sel)) AND NOT (fb_0.S_Mode5Sel)) AND NOT (fb_0.S_Mode6Sel)) AND NOT (fb_0.S_Mode7Sel)));
	testState_0 := testState_0 + 1;
35:
	fb_0.Activate := TRUE; fb_0.AutoSetMode := TRUE; fb_0.S_SetMode := FALSE; fb_0.S_Unlock := FALSE; fb_0.Reset := FALSE; fb_0.S_Mode0 := FALSE; fb_0.S_Mode1 := TRUE; fb_0.S_Mode2 := FALSE; fb_0.S_Mode3 := FALSE; fb_0.S_Mode4 := FALSE; fb_0.S_Mode5 := FALSE; fb_0.S_Mode6 := FALSE; fb_0.S_Mode7 := FALSE;
	fb_0();
	failed_0 := NOT (((((((((((((((((NOT (fb_0.Reset_Before) AND NOT (fb_0.S_SetMode_Before)) AND NOT (fb_0.T_1.Q)) AND (fb_0.DiagCode = 32784)) AND fb_0.Ready) AND NOT (fb_0.SafetyDemand)) AND NOT (fb_0.ResetRequest)) AND NOT (fb_0.Error)) AND fb_0.S_AnyModeSel) AND NOT (fb_0.S_Mode0Sel)) AND fb_0.S_Mode1Sel) AND NOT (fb_0.S_Mode2Sel)) AND NOT (fb_0.S_Mode3Sel)) AND NOT (fb_0.S_Mode4Sel)) AND NOT (fb_0.S_Mode5Sel)) AND NOT (fb_0.S_Mode6Sel)) AND NOT (fb_0.S_Mode7Sel)));
	testState_0 := testState_0 + 1;
36:
	fb_0.Activate := TRUE; fb_0.AutoSetMode := TRUE; fb_0.S_SetMode := FALSE; fb_0.S_Unlock := FALSE; fb_0.Reset := FALSE; fb_0.S_Mode0 := FALSE; fb_0.S_Mode1 := TRUE; fb_0.S_Mode2 := FALSE; fb_0.S_Mode3 := FALSE; fb_0.S_Mode4 := FALSE; fb_0.S_Mode5 := FALSE; fb_0.S_Mode6 := FALSE; fb_0.S_Mode7 := FALSE;
	fb_0();
	failed_0 := NOT (((((((((((((((((NOT (fb_0.Reset_Before) AND NOT (fb_0.S_SetMode_Before)) AND NOT (fb_0.T_1.Q)) AND (fb_0.DiagCode = 32784)) AND fb_0.Ready) AND NOT (fb_0.SafetyDemand)) AND NOT (fb_0.ResetRequest)) AND NOT (fb_0.Error)) AND fb_0.S_AnyModeSel) AND NOT (fb_0.S_Mode0Sel)) AND fb_0.S_Mode1Sel) AND NOT (fb_0.S_Mode2Sel)) AND NOT (fb_0.S_Mode3Sel)) AND NOT (fb_0.S_Mode4Sel)) AND NOT (fb_0.S_Mode5Sel)) AND NOT (fb_0.S_Mode6Sel)) AND NOT (fb_0.S_Mode7Sel)));
	testState_0 := testState_0 + 1;
37:
	fb_0.Activate := TRUE; fb_0.AutoSetMode := TRUE; fb_0.S_SetMode := FALSE; fb_0.S_Unlock := TRUE; fb_0.Reset := FALSE; fb_0.S_Mode0 := FALSE; fb_0.S_Mode1 := TRUE; fb_0.S_Mode2 := FALSE; fb_0.S_Mode3 := FALSE; fb_0.S_Mode4 := FALSE; fb_0.S_Mode5 := FALSE; fb_0.S_Mode6 := FALSE; fb_0.S_Mode7 := FALSE;
	fb_0();
	failed_0 := NOT (((((((((((((((((NOT (fb_0.Reset_Before) AND NOT (fb_0.S_SetMode_Before)) AND NOT (fb_0.T_1.Q)) AND (fb_0.DiagCode = 32768)) AND fb_0.Ready) AND NOT (fb_0.SafetyDemand)) AND NOT (fb_0.ResetRequest)) AND NOT (fb_0.Error)) AND fb_0.S_AnyModeSel) AND NOT (fb_0.S_Mode0Sel)) AND fb_0.S_Mode1Sel) AND NOT (fb_0.S_Mode2Sel)) AND NOT (fb_0.S_Mode3Sel)) AND NOT (fb_0.S_Mode4Sel)) AND NOT (fb_0.S_Mode5Sel)) AND NOT (fb_0.S_Mode6Sel)) AND NOT (fb_0.S_Mode7Sel)));
	testState_0 := testState_0 + 1;
38:
	fb_0.Activate := TRUE; fb_0.AutoSetMode := TRUE; fb_0.S_SetMode := FALSE; fb_0.S_Unlock := TRUE; fb_0.Reset := FALSE; fb_0.S_Mode0 := FALSE; fb_0.S_Mode1 := TRUE; fb_0.S_Mode2 := FALSE; fb_0.S_Mode3 := FALSE; fb_0.S_Mode4 := FALSE; fb_0.S_Mode5 := FALSE; fb_0.S_Mode6 := FALSE; fb_0.S_Mode7 := FALSE;
	fb_0();
	failed_0 := NOT (((((((((((((((((NOT (fb_0.Reset_Before) AND NOT (fb_0.S_SetMode_Before)) AND NOT (fb_0.T_1.Q)) AND (fb_0.DiagCode = 32768)) AND fb_0.Ready) AND NOT (fb_0.SafetyDemand)) AND NOT (fb_0.ResetRequest)) AND NOT (fb_0.Error)) AND fb_0.S_AnyModeSel) AND NOT (fb_0.S_Mode0Sel)) AND fb_0.S_Mode1Sel) AND NOT (fb_0.S_Mode2Sel)) AND NOT (fb_0.S_Mode3Sel)) AND NOT (fb_0.S_Mode4Sel)) AND NOT (fb_0.S_Mode5Sel)) AND NOT (fb_0.S_Mode6Sel)) AND NOT (fb_0.S_Mode7Sel)));
	testState_0 := testState_0 + 1;
39:
	fb_0.Activate := TRUE; fb_0.AutoSetMode := TRUE; fb_0.S_SetMode := FALSE; fb_0.S_Unlock := FALSE; fb_0.Reset := FALSE; fb_0.S_Mode0 := FALSE; fb_0.S_Mode1 := FALSE; fb_0.S_Mode2 := FALSE; fb_0.S_Mode3 := FALSE; fb_0.S_Mode4 := FALSE; fb_0.S_Mode5 := FALSE; fb_0.S_Mode6 := FALSE; fb_0.S_Mode7 := FALSE;
	fb_0();
	failed_0 := NOT (((((((((((((((((NOT (fb_0.Reset_Before) AND NOT (fb_0.S_SetMode_Before)) AND NOT (fb_0.T_1.Q)) AND (fb_0.DiagCode = 34818)) AND fb_0.Ready) AND fb_0.SafetyDemand) AND NOT (fb_0.ResetRequest)) AND NOT (fb_0.Error)) AND NOT (fb_0.S_AnyModeSel)) AND NOT (fb_0.S_Mode0Sel)) AND NOT (fb_0.S_Mode1Sel)) AND NOT (fb_0.S_Mode2Sel)) AND NOT (fb_0.S_Mode3Sel)) AND NOT (fb_0.S_Mode4Sel)) AND NOT (fb_0.S_Mode5Sel)) AND NOT (fb_0.S_Mode6Sel)) AND NOT (fb_0.S_Mode7Sel)));
	testState_0 := testState_0 + 1;
40:
	fb_0.Activate := TRUE; fb_0.AutoSetMode := TRUE; fb_0.S_SetMode := FALSE; fb_0.S_Unlock := TRUE; fb_0.Reset := FALSE; fb_0.S_Mode0 := FALSE; fb_0.S_Mode1 := FALSE; fb_0.S_Mode2 := TRUE; fb_0.S_Mode3 := FALSE; fb_0.S_Mode4 := FALSE; fb_0.S_Mode5 := FALSE; fb_0.S_Mode6 := FALSE; fb_0.S_Mode7 := FALSE;
	fb_0();
	failed_0 := NOT (((((((((((((((((NOT (fb_0.Reset_Before) AND NOT (fb_0.S_SetMode_Before)) AND NOT (fb_0.T_1.Q)) AND (fb_0.DiagCode = 32768)) AND fb_0.Ready) AND NOT (fb_0.SafetyDemand)) AND NOT (fb_0.ResetRequest)) AND NOT (fb_0.Error)) AND fb_0.S_AnyModeSel) AND NOT (fb_0.S_Mode0Sel)) AND NOT (fb_0.S_Mode1Sel)) AND fb_0.S_Mode2Sel) AND NOT (fb_0.S_Mode3Sel)) AND NOT (fb_0.S_Mode4Sel)) AND NOT (fb_0.S_Mode5Sel)) AND NOT (fb_0.S_Mode6Sel)) AND NOT (fb_0.S_Mode7Sel)));
	testState_0 := testState_0 + 1;
41:
	fb_0.Activate := TRUE; fb_0.AutoSetMode := TRUE; fb_0.S_SetMode := FALSE; fb_0.S_Unlock := FALSE; fb_0.Reset := FALSE; fb_0.S_Mode0 := FALSE; fb_0.S_Mode1 := FALSE; fb_0.S_Mode2 := TRUE; fb_0.S_Mode3 := FALSE; fb_0.S_Mode4 := FALSE; fb_0.S_Mode5 := FALSE; fb_0.S_Mode6 := FALSE; fb_0.S_Mode7 := FALSE;
	fb_0();
	failed_0 := NOT (((((((((((((((((NOT (fb_0.Reset_Before) AND NOT (fb_0.S_SetMode_Before)) AND NOT (fb_0.T_1.Q)) AND (fb_0.DiagCode = 32784)) AND fb_0.Ready) AND NOT (fb_0.SafetyDemand)) AND NOT (fb_0.ResetRequest)) AND NOT (fb_0.Error)) AND fb_0.S_AnyModeSel) AND NOT (fb_0.S_Mode0Sel)) AND NOT (fb_0.S_Mode1Sel)) AND fb_0.S_Mode2Sel) AND NOT (fb_0.S_Mode3Sel)) AND NOT (fb_0.S_Mode4Sel)) AND NOT (fb_0.S_Mode5Sel)) AND NOT (fb_0.S_Mode6Sel)) AND NOT (fb_0.S_Mode7Sel)));
	testState_0 := testState_0 + 1;
42:
	fb_0.Activate := TRUE; fb_0.AutoSetMode := TRUE; fb_0.S_SetMode := FALSE; fb_0.S_Unlock := TRUE; fb_0.Reset := FALSE; fb_0.S_Mode0 := FALSE; fb_0.S_Mode1 := FALSE; fb_0.S_Mode2 := FALSE; fb_0.S_Mode3 := FALSE; fb_0.S_Mode4 := FALSE; fb_0.S_Mode5 := FALSE; fb_0.S_Mode6 := FALSE; fb_0.S_Mode7 := FALSE;
	fb_0();
	failed_0 := NOT (((((((((((((((((NOT (fb_0.Reset_Before) AND NOT (fb_0.S_SetMode_Before)) AND NOT (fb_0.T_1.Q)) AND (fb_0.DiagCode = 34818)) AND fb_0.Ready) AND fb_0.SafetyDemand) AND NOT (fb_0.ResetRequest)) AND NOT (fb_0.Error)) AND NOT (fb_0.S_AnyModeSel)) AND NOT (fb_0.S_Mode0Sel)) AND NOT (fb_0.S_Mode1Sel)) AND NOT (fb_0.S_Mode2Sel)) AND NOT (fb_0.S_Mode3Sel)) AND NOT (fb_0.S_Mode4Sel)) AND NOT (fb_0.S_Mode5Sel)) AND NOT (fb_0.S_Mode6Sel)) AND NOT (fb_0.S_Mode7Sel)));
	testState_0 := testState_0 + 1;
43:
	fb_0.Activate := TRUE; fb_0.AutoSetMode := TRUE; fb_0.S_SetMode := FALSE; fb_0.S_Unlock := TRUE; fb_0.Reset := FALSE; fb_0.S_Mode0 := FALSE; fb_0.S_Mode1 := FALSE; fb_0.S_Mode2 := FALSE; fb_0.S_Mode3 := TRUE; fb_0.S_Mode4 := FALSE; fb_0.S_Mode5 := FALSE; fb_0.S_Mode6 := FALSE; fb_0.S_Mode7 := FALSE;
	fb_0();
	failed_0 := NOT (((((((((((((((((NOT (fb_0.Reset_Before) AND NOT (fb_0.S_SetMode_Before)) AND NOT (fb_0.T_1.Q)) AND (fb_0.DiagCode = 32768)) AND fb_0.Ready) AND NOT (fb_0.SafetyDemand)) AND NOT (fb_0.ResetRequest)) AND NOT (fb_0.Error)) AND fb_0.S_AnyModeSel) AND NOT (fb_0.S_Mode0Sel)) AND NOT (fb_0.S_Mode1Sel)) AND NOT (fb_0.S_Mode2Sel)) AND fb_0.S_Mode3Sel) AND NOT (fb_0.S_Mode4Sel)) AND NOT (fb_0.S_Mode5Sel)) AND NOT (fb_0.S_Mode6Sel)) AND NOT (fb_0.S_Mode7Sel)));
	testState_0 := testState_0 + 1;
44:
	fb_0.Activate := TRUE; fb_0.AutoSetMode := TRUE; fb_0.S_SetMode := FALSE; fb_0.S_Unlock := FALSE; fb_0.Reset := FALSE; fb_0.S_Mode0 := FALSE; fb_0.S_Mode1 := FALSE; fb_0.S_Mode2 := FALSE; fb_0.S_Mode3 := TRUE; fb_0.S_Mode4 := TRUE; fb_0.S_Mode5 := FALSE; fb_0.S_Mode6 := FALSE; fb_0.S_Mode7 := FALSE;
	fb_0();
	failed_0 := NOT (((((((((((((((((NOT (fb_0.Reset_Before) AND NOT (fb_0.S_SetMode_Before)) AND NOT (fb_0.T_1.Q)) AND (fb_0.DiagCode = 49168)) AND fb_0.Ready) AND NOT (fb_0.SafetyDemand)) AND NOT (fb_0.ResetRequest)) AND fb_0.Error) AND NOT (fb_0.S_AnyModeSel)) AND NOT (fb_0.S_Mode0Sel)) AND NOT (fb_0.S_Mode1Sel)) AND NOT (fb_0.S_Mode2Sel)) AND NOT (fb_0.S_Mode3Sel)) AND NOT (fb_0.S_Mode4Sel)) AND NOT (fb_0.S_Mode5Sel)) AND NOT (fb_0.S_Mode6Sel)) AND NOT (fb_0.S_Mode7Sel)));
	testState_0 := testState_0 + 1;
45:
	fb_0.Activate := TRUE; fb_0.AutoSetMode := TRUE; fb_0.S_SetMode := FALSE; fb_0.S_Unlock := FALSE; fb_0.Reset := TRUE; fb_0.S_Mode0 := FALSE; fb_0.S_Mode1 := FALSE; fb_0.S_Mode2 := FALSE; fb_0.S_Mode3 := FALSE; fb_0.S_Mode4 := FALSE; fb_0.S_Mode5 := FALSE; fb_0.S_Mode6 := FALSE; fb_0.S_Mode7 := FALSE;
	fb_0();
	failed_0 := NOT (((((((((((((((((fb_0.Reset_Before AND NOT (fb_0.S_SetMode_Before)) AND NOT (fb_0.T_1.Q)) AND (fb_0.DiagCode = 34818)) AND fb_0.Ready) AND fb_0.SafetyDemand) AND NOT (fb_0.ResetRequest)) AND NOT (fb_0.Error)) AND NOT (fb_0.S_AnyModeSel)) AND NOT (fb_0.S_Mode0Sel)) AND NOT (fb_0.S_Mode1Sel)) AND NOT (fb_0.S_Mode2Sel)) AND NOT (fb_0.S_Mode3Sel)) AND NOT (fb_0.S_Mode4Sel)) AND NOT (fb_0.S_Mode5Sel)) AND NOT (fb_0.S_Mode6Sel)) AND NOT (fb_0.S_Mode7Sel)));
	testState_0 := testState_0 + 1;
46:
	fb_0.Activate := TRUE; fb_0.AutoSetMode := TRUE; fb_0.S_SetMode := FALSE; fb_0.S_Unlock := TRUE; fb_0.Reset := FALSE; fb_0.S_Mode0 := FALSE; fb_0.S_Mode1 := FALSE; fb_0.S_Mode2 := FALSE; fb_0.S_Mode3 := TRUE; fb_0.S_Mode4 := FALSE; fb_0.S_Mode5 := FALSE; fb_0.S_Mode6 := FALSE; fb_0.S_Mode7 := FALSE;
	fb_0();
	failed_0 := NOT (((((((((((((((((NOT (fb_0.Reset_Before) AND NOT (fb_0.S_SetMode_Before)) AND NOT (fb_0.T_1.Q)) AND (fb_0.DiagCode = 32768)) AND fb_0.Ready) AND NOT (fb_0.SafetyDemand)) AND NOT (fb_0.ResetRequest)) AND NOT (fb_0.Error)) AND fb_0.S_AnyModeSel) AND NOT (fb_0.S_Mode0Sel)) AND NOT (fb_0.S_Mode1Sel)) AND NOT (fb_0.S_Mode2Sel)) AND fb_0.S_Mode3Sel) AND NOT (fb_0.S_Mode4Sel)) AND NOT (fb_0.S_Mode5Sel)) AND NOT (fb_0.S_Mode6Sel)) AND NOT (fb_0.S_Mode7Sel)));
	testState_0 := testState_0 + 1;
47:
	fb_0.Activate := TRUE; fb_0.AutoSetMode := TRUE; fb_0.S_SetMode := FALSE; fb_0.S_Unlock := FALSE; fb_0.Reset := FALSE; fb_0.S_Mode0 := FALSE; fb_0.S_Mode1 := FALSE; fb_0.S_Mode2 := FALSE; fb_0.S_Mode3 := TRUE; fb_0.S_Mode4 := FALSE; fb_0.S_Mode5 := FALSE; fb_0.S_Mode6 := FALSE; fb_0.S_Mode7 := FALSE;
	fb_0();
	failed_0 := NOT (((((((((((((((((NOT (fb_0.Reset_Before) AND NOT (fb_0.S_SetMode_Before)) AND NOT (fb_0.T_1.Q)) AND (fb_0.DiagCode = 32784)) AND fb_0.Ready) AND NOT (fb_0.SafetyDemand)) AND NOT (fb_0.ResetRequest)) AND NOT (fb_0.Error)) AND fb_0.S_AnyModeSel) AND NOT (fb_0.S_Mode0Sel)) AND NOT (fb_0.S_Mode1Sel)) AND NOT (fb_0.S_Mode2Sel)) AND fb_0.S_Mode3Sel) AND NOT (fb_0.S_Mode4Sel)) AND NOT (fb_0.S_Mode5Sel)) AND NOT (fb_0.S_Mode6Sel)) AND NOT (fb_0.S_Mode7Sel)));
	testState_0 := testState_0 + 1;
48:
	fb_0.Activate := TRUE; fb_0.AutoSetMode := TRUE; fb_0.S_SetMode := FALSE; fb_0.S_Unlock := TRUE; fb_0.Reset := FALSE; fb_0.S_Mode0 := FALSE; fb_0.S_Mode1 := FALSE; fb_0.S_Mode2 := FALSE; fb_0.S_Mode3 := TRUE; fb_0.S_Mode4 := FALSE; fb_0.S_Mode5 := FALSE; fb_0.S_Mode6 := FALSE; fb_0.S_Mode7 := FALSE;
	fb_0();
	failed_0 := NOT (((((((((((((((((NOT (fb_0.Reset_Before) AND NOT (fb_0.S_SetMode_Before)) AND NOT (fb_0.T_1.Q)) AND (fb_0.DiagCode = 32768)) AND fb_0.Ready) AND NOT (fb_0.SafetyDemand)) AND NOT (fb_0.ResetRequest)) AND NOT (fb_0.Error)) AND fb_0.S_AnyModeSel) AND NOT (fb_0.S_Mode0Sel)) AND NOT (fb_0.S_Mode1Sel)) AND NOT (fb_0.S_Mode2Sel)) AND fb_0.S_Mode3Sel) AND NOT (fb_0.S_Mode4Sel)) AND NOT (fb_0.S_Mode5Sel)) AND NOT (fb_0.S_Mode6Sel)) AND NOT (fb_0.S_Mode7Sel)));
	testState_0 := testState_0 + 1;
49:
	fb_0.Activate := TRUE; fb_0.AutoSetMode := TRUE; fb_0.S_SetMode := FALSE; fb_0.S_Unlock := FALSE; fb_0.Reset := FALSE; fb_0.S_Mode0 := FALSE; fb_0.S_Mode1 := FALSE; fb_0.S_Mode2 := FALSE; fb_0.S_Mode3 := FALSE; fb_0.S_Mode4 := FALSE; fb_0.S_Mode5 := FALSE; fb_0.S_Mode6 := FALSE; fb_0.S_Mode7 := FALSE;
	fb_0();
	failed_0 := NOT (((((((((((((((((NOT (fb_0.Reset_Before) AND NOT (fb_0.S_SetMode_Before)) AND NOT (fb_0.T_1.Q)) AND (fb_0.DiagCode = 34818)) AND fb_0.Ready) AND fb_0.SafetyDemand) AND NOT (fb_0.ResetRequest)) AND NOT (fb_0.Error)) AND NOT (fb_0.S_AnyModeSel)) AND NOT (fb_0.S_Mode0Sel)) AND NOT (fb_0.S_Mode1Sel)) AND NOT (fb_0.S_Mode2Sel)) AND NOT (fb_0.S_Mode3Sel)) AND NOT (fb_0.S_Mode4Sel)) AND NOT (fb_0.S_Mode5Sel)) AND NOT (fb_0.S_Mode6Sel)) AND NOT (fb_0.S_Mode7Sel)));
	testState_0 := testState_0 + 1;
50:
	fb_0.Activate := TRUE; fb_0.AutoSetMode := TRUE; fb_0.S_SetMode := FALSE; fb_0.S_Unlock := TRUE; fb_0.Reset := FALSE; fb_0.S_Mode0 := FALSE; fb_0.S_Mode1 := FALSE; fb_0.S_Mode2 := FALSE; fb_0.S_Mode3 := FALSE; fb_0.S_Mode4 := TRUE; fb_0.S_Mode5 := FALSE; fb_0.S_Mode6 := FALSE; fb_0.S_Mode7 := FALSE;
	fb_0();
	failed_0 := NOT (((((((((((((((((NOT (fb_0.Reset_Before) AND NOT (fb_0.S_SetMode_Before)) AND NOT (fb_0.T_1.Q)) AND (fb_0.DiagCode = 32768)) AND fb_0.Ready) AND NOT (fb_0.SafetyDemand)) AND NOT (fb_0.ResetRequest)) AND NOT (fb_0.Error)) AND fb_0.S_AnyModeSel) AND NOT (fb_0.S_Mode0Sel)) AND NOT (fb_0.S_Mode1Sel)) AND NOT (fb_0.S_Mode2Sel)) AND NOT (fb_0.S_Mode3Sel)) AND fb_0.S_Mode4Sel) AND NOT (fb_0.S_Mode5Sel)) AND NOT (fb_0.S_Mode6Sel)) AND NOT (fb_0.S_Mode7Sel)));
	testState_0 := testState_0 + 1;
51:
	fb_0.Activate := TRUE; fb_0.AutoSetMode := TRUE; fb_0.S_SetMode := FALSE; fb_0.S_Unlock := FALSE; fb_0.Reset := FALSE; fb_0.S_Mode0 := FALSE; fb_0.S_Mode1 := FALSE; fb_0.S_Mode2 := FALSE; fb_0.S_Mode3 := FALSE; fb_0.S_Mode4 := TRUE; fb_0.S_Mode5 := FALSE; fb_0.S_Mode6 := FALSE; fb_0.S_Mode7 := FALSE;
	fb_0();
	failed_0 := NOT (((((((((((((((((NOT (fb_0.Reset_Before) AND NOT (fb_0.S_SetMode_Before)) AND NOT (fb_0.T_1.Q)) AND (fb_0.DiagCode = 32784)) AND fb_0.Ready) AND NOT (fb_0.SafetyDemand)) AND NOT (fb_0.ResetRequest)) AND NOT (fb_0.Error)) AND fb_0.S_AnyModeSel) AND NOT (fb_0.S_Mode0Sel)) AND NOT (fb_0.S_Mode1Sel)) AND NOT (fb_0.S_Mode2Sel)) AND NOT (fb_0.S_Mode3Sel)) AND fb_0.S_Mode4Sel) AND NOT (fb_0.S_Mode5Sel)) AND NOT (fb_0.S_Mode6Sel)) AND NOT (fb_0.S_Mode7Sel)));
	testState_0 := testState_0 + 1;
52:
	fb_0.Activate := TRUE; fb_0.AutoSetMode := TRUE; fb_0.S_SetMode := FALSE; fb_0.S_Unlock := TRUE; fb_0.Reset := FALSE; fb_0.S_Mode0 := FALSE; fb_0.S_Mode1 := FALSE; fb_0.S_Mode2 := FALSE; fb_0.S_Mode3 := FALSE; fb_0.S_Mode4 := TRUE; fb_0.S_Mode5 := TRUE; fb_0.S_Mode6 := FALSE; fb_0.S_Mode7 := FALSE;
	fb_0();
	failed_0 := NOT (((((((((((((((((NOT (fb_0.Reset_Before) AND NOT (fb_0.S_SetMode_Before)) AND NOT (fb_0.T_1.Q)) AND (fb_0.DiagCode = 49168)) AND fb_0.Ready) AND NOT (fb_0.SafetyDemand)) AND NOT (fb_0.ResetRequest)) AND fb_0.Error) AND NOT (fb_0.S_AnyModeSel)) AND NOT (fb_0.S_Mode0Sel)) AND NOT (fb_0.S_Mode1Sel)) AND NOT (fb_0.S_Mode2Sel)) AND NOT (fb_0.S_Mode3Sel)) AND NOT (fb_0.S_Mode4Sel)) AND NOT (fb_0.S_Mode5Sel)) AND NOT (fb_0.S_Mode6Sel)) AND NOT (fb_0.S_Mode7Sel)));
	testState_0 := testState_0 + 1;
53:
	fb_0.Activate := TRUE; fb_0.AutoSetMode := TRUE; fb_0.S_SetMode := FALSE; fb_0.S_Unlock := FALSE; fb_0.Reset := TRUE; fb_0.S_Mode0 := FALSE; fb_0.S_Mode1 := FALSE; fb_0.S_Mode2 := FALSE; fb_0.S_Mode3 := FALSE; fb_0.S_Mode4 := FALSE; fb_0.S_Mode5 := FALSE; fb_0.S_Mode6 := FALSE; fb_0.S_Mode7 := FALSE;
	fb_0();
	failed_0 := NOT (((((((((((((((((fb_0.Reset_Before AND NOT (fb_0.S_SetMode_Before)) AND NOT (fb_0.T_1.Q)) AND (fb_0.DiagCode = 34818)) AND fb_0.Ready) AND fb_0.SafetyDemand) AND NOT (fb_0.ResetRequest)) AND NOT (fb_0.Error)) AND NOT (fb_0.S_AnyModeSel)) AND NOT (fb_0.S_Mode0Sel)) AND NOT (fb_0.S_Mode1Sel)) AND NOT (fb_0.S_Mode2Sel)) AND NOT (fb_0.S_Mode3Sel)) AND NOT (fb_0.S_Mode4Sel)) AND NOT (fb_0.S_Mode5Sel)) AND NOT (fb_0.S_Mode6Sel)) AND NOT (fb_0.S_Mode7Sel)));
	testState_0 := testState_0 + 1;
54:
	fb_0.Activate := TRUE; fb_0.AutoSetMode := TRUE; fb_0.S_SetMode := FALSE; fb_0.S_Unlock := TRUE; fb_0.Reset := FALSE; fb_0.S_Mode0 := FALSE; fb_0.S_Mode1 := FALSE; fb_0.S_Mode2 := FALSE; fb_0.S_Mode3 := FALSE; fb_0.S_Mode4 := FALSE; fb_0.S_Mode5 := TRUE; fb_0.S_Mode6 := FALSE; fb_0.S_Mode7 := FALSE;
	fb_0();
	failed_0 := NOT (((((((((((((((((NOT (fb_0.Reset_Before) AND NOT (fb_0.S_SetMode_Before)) AND NOT (fb_0.T_1.Q)) AND (fb_0.DiagCode = 32768)) AND fb_0.Ready) AND NOT (fb_0.SafetyDemand)) AND NOT (fb_0.ResetRequest)) AND NOT (fb_0.Error)) AND fb_0.S_AnyModeSel) AND NOT (fb_0.S_Mode0Sel)) AND NOT (fb_0.S_Mode1Sel)) AND NOT (fb_0.S_Mode2Sel)) AND NOT (fb_0.S_Mode3Sel)) AND NOT (fb_0.S_Mode4Sel)) AND fb_0.S_Mode5Sel) AND NOT (fb_0.S_Mode6Sel)) AND NOT (fb_0.S_Mode7Sel)));
	testState_0 := testState_0 + 1;
55:
	fb_0.Activate := TRUE; fb_0.AutoSetMode := TRUE; fb_0.S_SetMode := FALSE; fb_0.S_Unlock := FALSE; fb_0.Reset := FALSE; fb_0.S_Mode0 := FALSE; fb_0.S_Mode1 := FALSE; fb_0.S_Mode2 := FALSE; fb_0.S_Mode3 := FALSE; fb_0.S_Mode4 := FALSE; fb_0.S_Mode5 := TRUE; fb_0.S_Mode6 := FALSE; fb_0.S_Mode7 := FALSE;
	fb_0();
	failed_0 := NOT (((((((((((((((((NOT (fb_0.Reset_Before) AND NOT (fb_0.S_SetMode_Before)) AND NOT (fb_0.T_1.Q)) AND (fb_0.DiagCode = 32784)) AND fb_0.Ready) AND NOT (fb_0.SafetyDemand)) AND NOT (fb_0.ResetRequest)) AND NOT (fb_0.Error)) AND fb_0.S_AnyModeSel) AND NOT (fb_0.S_Mode0Sel)) AND NOT (fb_0.S_Mode1Sel)) AND NOT (fb_0.S_Mode2Sel)) AND NOT (fb_0.S_Mode3Sel)) AND NOT (fb_0.S_Mode4Sel)) AND fb_0.S_Mode5Sel) AND NOT (fb_0.S_Mode6Sel)) AND NOT (fb_0.S_Mode7Sel)));
	testState_0 := testState_0 + 1;
56:
	fb_0.Activate := TRUE; fb_0.AutoSetMode := TRUE; fb_0.S_SetMode := FALSE; fb_0.S_Unlock := TRUE; fb_0.Reset := FALSE; fb_0.S_Mode0 := FALSE; fb_0.S_Mode1 := FALSE; fb_0.S_Mode2 := FALSE; fb_0.S_Mode3 := FALSE; fb_0.S_Mode4 := FALSE; fb_0.S_Mode5 := TRUE; fb_0.S_Mode6 := FALSE; fb_0.S_Mode7 := FALSE;
	fb_0();
	failed_0 := NOT (((((((((((((((((NOT (fb_0.Reset_Before) AND NOT (fb_0.S_SetMode_Before)) AND NOT (fb_0.T_1.Q)) AND (fb_0.DiagCode = 32768)) AND fb_0.Ready) AND NOT (fb_0.SafetyDemand)) AND NOT (fb_0.ResetRequest)) AND NOT (fb_0.Error)) AND fb_0.S_AnyModeSel) AND NOT (fb_0.S_Mode0Sel)) AND NOT (fb_0.S_Mode1Sel)) AND NOT (fb_0.S_Mode2Sel)) AND NOT (fb_0.S_Mode3Sel)) AND NOT (fb_0.S_Mode4Sel)) AND fb_0.S_Mode5Sel) AND NOT (fb_0.S_Mode6Sel)) AND NOT (fb_0.S_Mode7Sel)));
	testState_0 := testState_0 + 1;
57:
	fb_0.Activate := TRUE; fb_0.AutoSetMode := TRUE; fb_0.S_SetMode := FALSE; fb_0.S_Unlock := FALSE; fb_0.Reset := FALSE; fb_0.S_Mode0 := FALSE; fb_0.S_Mode1 := FALSE; fb_0.S_Mode2 := FALSE; fb_0.S_Mode3 := FALSE; fb_0.S_Mode4 := FALSE; fb_0.S_Mode5 := FALSE; fb_0.S_Mode6 := FALSE; fb_0.S_Mode7 := FALSE;
	fb_0();
	failed_0 := NOT (((((((((((((((((NOT (fb_0.Reset_Before) AND NOT (fb_0.S_SetMode_Before)) AND NOT (fb_0.T_1.Q)) AND (fb_0.DiagCode = 34818)) AND fb_0.Ready) AND fb_0.SafetyDemand) AND NOT (fb_0.ResetRequest)) AND NOT (fb_0.Error)) AND NOT (fb_0.S_AnyModeSel)) AND NOT (fb_0.S_Mode0Sel)) AND NOT (fb_0.S_Mode1Sel)) AND NOT (fb_0.S_Mode2Sel)) AND NOT (fb_0.S_Mode3Sel)) AND NOT (fb_0.S_Mode4Sel)) AND NOT (fb_0.S_Mode5Sel)) AND NOT (fb_0.S_Mode6Sel)) AND NOT (fb_0.S_Mode7Sel)));
	testState_0 := testState_0 + 1;
58:
	fb_0.Activate := TRUE; fb_0.AutoSetMode := TRUE; fb_0.S_SetMode := FALSE; fb_0.S_Unlock := TRUE; fb_0.Reset := FALSE; fb_0.S_Mode0 := FALSE; fb_0.S_Mode1 := FALSE; fb_0.S_Mode2 := FALSE; fb_0.S_Mode3 := FALSE; fb_0.S_Mode4 := FALSE; fb_0.S_Mode5 := FALSE; fb_0.S_Mode6 := TRUE; fb_0.S_Mode7 := FALSE;
	fb_0();
	failed_0 := NOT (((((((((((((((((NOT (fb_0.Reset_Before) AND NOT (fb_0.S_SetMode_Before)) AND NOT (fb_0.T_1.Q)) AND (fb_0.DiagCode = 32768)) AND fb_0.Ready) AND NOT (fb_0.SafetyDemand)) AND NOT (fb_0.ResetRequest)) AND NOT (fb_0.Error)) AND fb_0.S_AnyModeSel) AND NOT (fb_0.S_Mode0Sel)) AND NOT (fb_0.S_Mode1Sel)) AND NOT (fb_0.S_Mode2Sel)) AND NOT (fb_0.S_Mode3Sel)) AND NOT (fb_0.S_Mode4Sel)) AND NOT (fb_0.S_Mode5Sel)) AND fb_0.S_Mode6Sel) AND NOT (fb_0.S_Mode7Sel)));
	testState_0 := testState_0 + 1;
59:
	fb_0.Activate := TRUE; fb_0.AutoSetMode := TRUE; fb_0.S_SetMode := FALSE; fb_0.S_Unlock := FALSE; fb_0.Reset := FALSE; fb_0.S_Mode0 := FALSE; fb_0.S_Mode1 := FALSE; fb_0.S_Mode2 := FALSE; fb_0.S_Mode3 := FALSE; fb_0.S_Mode4 := FALSE; fb_0.S_Mode5 := FALSE; fb_0.S_Mode6 := TRUE; fb_0.S_Mode7 := FALSE;
	fb_0();
	failed_0 := NOT (((((((((((((((((NOT (fb_0.Reset_Before) AND NOT (fb_0.S_SetMode_Before)) AND NOT (fb_0.T_1.Q)) AND (fb_0.DiagCode = 32784)) AND fb_0.Ready) AND NOT (fb_0.SafetyDemand)) AND NOT (fb_0.ResetRequest)) AND NOT (fb_0.Error)) AND fb_0.S_AnyModeSel) AND NOT (fb_0.S_Mode0Sel)) AND NOT (fb_0.S_Mode1Sel)) AND NOT (fb_0.S_Mode2Sel)) AND NOT (fb_0.S_Mode3Sel)) AND NOT (fb_0.S_Mode4Sel)) AND NOT (fb_0.S_Mode5Sel)) AND fb_0.S_Mode6Sel) AND NOT (fb_0.S_Mode7Sel)));
	testState_0 := testState_0 + 1;
60:
	fb_0.Activate := TRUE; fb_0.AutoSetMode := TRUE; fb_0.S_SetMode := FALSE; fb_0.S_Unlock := TRUE; fb_0.Reset := FALSE; fb_0.S_Mode0 := FALSE; fb_0.S_Mode1 := FALSE; fb_0.S_Mode2 := FALSE; fb_0.S_Mode3 := FALSE; fb_0.S_Mode4 := FALSE; fb_0.S_Mode5 := FALSE; fb_0.S_Mode6 := TRUE; fb_0.S_Mode7 := FALSE;
	fb_0();
	failed_0 := NOT (((((((((((((((((NOT (fb_0.Reset_Before) AND NOT (fb_0.S_SetMode_Before)) AND NOT (fb_0.T_1.Q)) AND (fb_0.DiagCode = 32768)) AND fb_0.Ready) AND NOT (fb_0.SafetyDemand)) AND NOT (fb_0.ResetRequest)) AND NOT (fb_0.Error)) AND fb_0.S_AnyModeSel) AND NOT (fb_0.S_Mode0Sel)) AND NOT (fb_0.S_Mode1Sel)) AND NOT (fb_0.S_Mode2Sel)) AND NOT (fb_0.S_Mode3Sel)) AND NOT (fb_0.S_Mode4Sel)) AND NOT (fb_0.S_Mode5Sel)) AND fb_0.S_Mode6Sel) AND NOT (fb_0.S_Mode7Sel)));
	testState_0 := testState_0 + 1;
61:
	fb_0.Activate := TRUE; fb_0.AutoSetMode := TRUE; fb_0.S_SetMode := FALSE; fb_0.S_Unlock := FALSE; fb_0.Reset := FALSE; fb_0.S_Mode0 := FALSE; fb_0.S_Mode1 := FALSE; fb_0.S_Mode2 := FALSE; fb_0.S_Mode3 := FALSE; fb_0.S_Mode4 := FALSE; fb_0.S_Mode5 := FALSE; fb_0.S_Mode6 := FALSE; fb_0.S_Mode7 := FALSE;
	fb_0();
	failed_0 := NOT (((((((((((((((((NOT (fb_0.Reset_Before) AND NOT (fb_0.S_SetMode_Before)) AND NOT (fb_0.T_1.Q)) AND (fb_0.DiagCode = 34818)) AND fb_0.Ready) AND fb_0.SafetyDemand) AND NOT (fb_0.ResetRequest)) AND NOT (fb_0.Error)) AND NOT (fb_0.S_AnyModeSel)) AND NOT (fb_0.S_Mode0Sel)) AND NOT (fb_0.S_Mode1Sel)) AND NOT (fb_0.S_Mode2Sel)) AND NOT (fb_0.S_Mode3Sel)) AND NOT (fb_0.S_Mode4Sel)) AND NOT (fb_0.S_Mode5Sel)) AND NOT (fb_0.S_Mode6Sel)) AND NOT (fb_0.S_Mode7Sel)));
	testState_0 := testState_0 + 1;
62:
	fb_0.Activate := TRUE; fb_0.AutoSetMode := TRUE; fb_0.S_SetMode := FALSE; fb_0.S_Unlock := TRUE; fb_0.Reset := FALSE; fb_0.S_Mode0 := FALSE; fb_0.S_Mode1 := FALSE; fb_0.S_Mode2 := FALSE; fb_0.S_Mode3 := FALSE; fb_0.S_Mode4 := FALSE; fb_0.S_Mode5 := FALSE; fb_0.S_Mode6 := FALSE; fb_0.S_Mode7 := TRUE;
	fb_0();
	failed_0 := NOT (((((((((((((((((NOT (fb_0.Reset_Before) AND NOT (fb_0.S_SetMode_Before)) AND NOT (fb_0.T_1.Q)) AND (fb_0.DiagCode = 32768)) AND fb_0.Ready) AND NOT (fb_0.SafetyDemand)) AND NOT (fb_0.ResetRequest)) AND NOT (fb_0.Error)) AND fb_0.S_AnyModeSel) AND NOT (fb_0.S_Mode0Sel)) AND NOT (fb_0.S_Mode1Sel)) AND NOT (fb_0.S_Mode2Sel)) AND NOT (fb_0.S_Mode3Sel)) AND NOT (fb_0.S_Mode4Sel)) AND NOT (fb_0.S_Mode5Sel)) AND NOT (fb_0.S_Mode6Sel)) AND fb_0.S_Mode7Sel));
	testState_0 := testState_0 + 1;
63:
	fb_0.Activate := TRUE; fb_0.AutoSetMode := TRUE; fb_0.S_SetMode := FALSE; fb_0.S_Unlock := FALSE; fb_0.Reset := FALSE; fb_0.S_Mode0 := FALSE; fb_0.S_Mode1 := FALSE; fb_0.S_Mode2 := FALSE; fb_0.S_Mode3 := FALSE; fb_0.S_Mode4 := FALSE; fb_0.S_Mode5 := FALSE; fb_0.S_Mode6 := FALSE; fb_0.S_Mode7 := TRUE;
	fb_0();
	failed_0 := NOT (((((((((((((((((NOT (fb_0.Reset_Before) AND NOT (fb_0.S_SetMode_Before)) AND NOT (fb_0.T_1.Q)) AND (fb_0.DiagCode = 32784)) AND fb_0.Ready) AND NOT (fb_0.SafetyDemand)) AND NOT (fb_0.ResetRequest)) AND NOT (fb_0.Error)) AND fb_0.S_AnyModeSel) AND NOT (fb_0.S_Mode0Sel)) AND NOT (fb_0.S_Mode1Sel)) AND NOT (fb_0.S_Mode2Sel)) AND NOT (fb_0.S_Mode3Sel)) AND NOT (fb_0.S_Mode4Sel)) AND NOT (fb_0.S_Mode5Sel)) AND NOT (fb_0.S_Mode6Sel)) AND fb_0.S_Mode7Sel));
	testState_0 := testState_0 + 1;
64:
	fb_0.Activate := TRUE; fb_0.AutoSetMode := TRUE; fb_0.S_SetMode := FALSE; fb_0.S_Unlock := TRUE; fb_0.Reset := FALSE; fb_0.S_Mode0 := FALSE; fb_0.S_Mode1 := FALSE; fb_0.S_Mode2 := FALSE; fb_0.S_Mode3 := FALSE; fb_0.S_Mode4 := FALSE; fb_0.S_Mode5 := FALSE; fb_0.S_Mode6 := FALSE; fb_0.S_Mode7 := TRUE;
	fb_0();
	failed_0 := NOT (((((((((((((((((NOT (fb_0.Reset_Before) AND NOT (fb_0.S_SetMode_Before)) AND NOT (fb_0.T_1.Q)) AND (fb_0.DiagCode = 32768)) AND fb_0.Ready) AND NOT (fb_0.SafetyDemand)) AND NOT (fb_0.ResetRequest)) AND NOT (fb_0.Error)) AND fb_0.S_AnyModeSel) AND NOT (fb_0.S_Mode0Sel)) AND NOT (fb_0.S_Mode1Sel)) AND NOT (fb_0.S_Mode2Sel)) AND NOT (fb_0.S_Mode3Sel)) AND NOT (fb_0.S_Mode4Sel)) AND NOT (fb_0.S_Mode5Sel)) AND NOT (fb_0.S_Mode6Sel)) AND fb_0.S_Mode7Sel));
	testState_0 := testState_0 + 1;
65:
	fb_0.Activate := TRUE; fb_0.AutoSetMode := TRUE; fb_0.S_SetMode := FALSE; fb_0.S_Unlock := FALSE; fb_0.Reset := FALSE; fb_0.S_Mode0 := FALSE; fb_0.S_Mode1 := FALSE; fb_0.S_Mode2 := FALSE; fb_0.S_Mode3 := FALSE; fb_0.S_Mode4 := FALSE; fb_0.S_Mode5 := FALSE; fb_0.S_Mode6 := FALSE; fb_0.S_Mode7 := FALSE;
	fb_0();
	failed_0 := NOT (((((((((((((((((NOT (fb_0.Reset_Before) AND NOT (fb_0.S_SetMode_Before)) AND NOT (fb_0.T_1.Q)) AND (fb_0.DiagCode = 34818)) AND fb_0.Ready) AND fb_0.SafetyDemand) AND NOT (fb_0.ResetRequest)) AND NOT (fb_0.Error)) AND NOT (fb_0.S_AnyModeSel)) AND NOT (fb_0.S_Mode0Sel)) AND NOT (fb_0.S_Mode1Sel)) AND NOT (fb_0.S_Mode2Sel)) AND NOT (fb_0.S_Mode3Sel)) AND NOT (fb_0.S_Mode4Sel)) AND NOT (fb_0.S_Mode5Sel)) AND NOT (fb_0.S_Mode6Sel)) AND NOT (fb_0.S_Mode7Sel)));
	testState_0 := testState_0 + 1;
66:
	fb_0.Activate := FALSE; fb_0.AutoSetMode := FALSE; fb_0.S_SetMode := FALSE; fb_0.S_Unlock := FALSE; fb_0.Reset := FALSE; fb_0.S_Mode0 := FALSE; fb_0.S_Mode1 := FALSE; fb_0.S_Mode2 := FALSE; fb_0.S_Mode3 := FALSE; fb_0.S_Mode4 := FALSE; fb_0.S_Mode5 := FALSE; fb_0.S_Mode6 := FALSE; fb_0.S_Mode7 := FALSE;
	fb_0();
	failed_0 := NOT ((NOT (fb_0.Reset_Before) AND (NOT (fb_0.S_SetMode_Before) AND (NOT (fb_0.T_1.Q) AND ((fb_0.DiagCode = 0) AND (NOT (fb_0.Ready) AND (NOT (fb_0.SafetyDemand) AND (NOT (fb_0.ResetRequest) AND (NOT (fb_0.Error) AND (NOT (fb_0.S_AnyModeSel) AND (NOT (fb_0.S_Mode0Sel) AND (NOT (fb_0.S_Mode1Sel) AND (NOT (fb_0.S_Mode2Sel) AND (NOT (fb_0.S_Mode3Sel) AND (NOT (fb_0.S_Mode4Sel) AND (NOT (fb_0.S_Mode5Sel) AND (NOT (fb_0.S_Mode6Sel) AND NOT (fb_0.S_Mode7Sel))))))))))))))))));
	testState_0 := testState_0 + 1;
67:
	finished_0 := TRUE;
END_CASE
END_IF

END_FUNCTION_BLOCK

(* ---- SF_TwoHandControlTypeII.st ---- *)
FUNCTION_BLOCK SF_TwoHandControlTypeII
VAR_INPUT
    Activate: BOOL;
    S_Button1: BOOL;
    S_Button2: BOOL;
END_VAR
VAR_OUTPUT
    Ready: BOOL;
    S_TwoHandOut: BOOL;
    SafetyDemand: BOOL;
    Error: BOOL;
    DiagCode: UINT;
END_VAR

BEGIN

IF NOT Activate THEN
    DiagCode := 16#0000;

    Ready := FALSE;
    SafetyDemand := FALSE;
    Error := FALSE;
    S_TwoHandOut := FALSE;

ELSE
    CASE DiagCode OF
    16#0000:
        DiagCode := 16#8001;
    16#8001:
        IF S_Button1 AND S_Button2 THEN
            DiagCode := 16#C030;
        ELSIF S_Button1 THEN
            DiagCode := 16#C010;
        ELSIF S_Button2 THEN
            DiagCode := 16#C020;
        ELSE
            DiagCode := 16#8802;
        END_IF;
    16#8802:
        IF S_Button1 AND S_Button2 THEN
            DiagCode := 16#8000;
        ELSIF S_Button1 THEN
            DiagCode := 16#8804;
        ELSIF S_Button2 THEN
            DiagCode := 16#8806;
        END_IF;
    16#8804:
        IF NOT (S_Button1 OR S_Button2) THEN
            DiagCode := 16#8802;
        ELSIF NOT S_Button1 AND S_Button2 THEN
            DiagCode := 16#880E;
        ELSIF S_Button1 AND S_Button2 THEN
            DiagCode := 16#8000;
        END_IF;
    16#8806:
        IF NOT (S_Button1 OR S_Button2) THEN
            DiagCode := 16#8802;
        ELSIF S_Button1 AND NOT S_Button2 THEN
            DiagCode := 16#880E;
        ELSIF S_Button1 AND S_Button2 THEN
            DiagCode := 16#8000;
        END_IF;
    16#8808:
        IF S_Button1 AND S_Button2 THEN
            DiagCode := 16#880C;
        ELSIF NOT S_Button1 AND S_Button2 THEN
            DiagCode := 16#880A;
        ELSIF NOT (S_Button1 OR S_Button2) THEN
            DiagCode := 16#8802;
        END_IF;
    16#880A:
        IF S_Button1 AND S_Button2 THEN
            DiagCode := 16#880C;
        ELSIF S_Button1 AND NOT S_Button2 THEN
            DiagCode := 16#8808;
        ELSIF NOT (S_Button1 OR S_Button2) THEN
            DiagCode := 16#8802;
        END_IF;
    16#880C:
        IF NOT S_Button1 AND S_Button2 THEN
            DiagCode := 16#880A;
        ELSIF S_Button1 AND NOT S_Button2 THEN
            DiagCode := 16#8808;
        ELSIF NOT (S_Button1 OR S_Button2) THEN
            DiagCode := 16#8802;
        END_IF;
    16#880E:
        IF NOT (S_Button1 OR S_Button2) THEN
            DiagCode := 16#8802;
        END_IF;
    16#8000:
        IF S_Button1 AND NOT S_Button2 THEN
            DiagCode := 16#8808;
        ELSIF NOT S_Button1 AND S_Button2 THEN
            DiagCode := 16#880A;
        ELSIF NOT (S_Button1 OR S_Button2) THEN
            DiagCode := 16#8802;
        END_IF;
    16#C010,
    16#C020,
    16#C030:
        IF NOT (S_Button1 OR S_Button2) THEN
            DiagCode := 16#8802;
        END_IF;
    END_CASE;

    CASE DiagCode OF
    16#8000:
        Ready := TRUE;
        SafetyDemand := FALSE;
        Error := FALSE;
        S_TwoHandOut := TRUE;
    16#8001:
        Ready := TRUE;
        SafetyDemand := FALSE;
        Error := FALSE;
        S_TwoHandOut := FALSE;
    16#8802,
    16#8804,
    16#8806,
    16#8808,
    16#880A,
    16#880C,
    16#880E:
        Ready := TRUE;
        SafetyDemand := TRUE;
        Error := FALSE;
        S_TwoHandOut := FALSE;
    16#C010,
    16#C020,
    16#C030:
        Ready := TRUE;
        SafetyDemand := FALSE;
        Error := TRUE;
        S_TwoHandOut := FALSE;
    END_CASE;
END_IF;

END_FUNCTION_BLOCK

(* ---- SF_TwoHandControlTypeII_Test.st ---- *)
FUNCTION_BLOCK SF_TwoHandControlTypeII_Test
VAR_INPUT
END_VAR
VAR_OUTPUT
	failed_0: BOOL := FALSE;
	finished_0: BOOL := FALSE;
END_VAR
VAR
	fb_0: SF_TwoHandControlTypeII_BranchCounters;
	waitCounter_0: UINT := 0;
	testState_0: UINT := 0;
END_VAR

IF NOT failed_0 AND NOT finished_0 THEN
CASE testState_0 OF
0:
	fb_0.Activate := FALSE;
	fb_0();
	failed_0 := NOT ((((((fb_0.DiagCode = 0) AND NOT (fb_0.Ready)) AND NOT (fb_0.S_TwoHandOut)) AND NOT (fb_0.SafetyDemand)) AND NOT (fb_0.Error)));
	testState_0 := testState_0 + 1;
1:
	fb_0.Activate := TRUE; fb_0.S_Button1 := FALSE; fb_0.S_Button2 := FALSE;
	fb_0();
	failed_0 := NOT ((((((fb_0.DiagCode = 32769) AND fb_0.Ready) AND NOT (fb_0.S_TwoHandOut)) AND NOT (fb_0.SafetyDemand)) AND NOT (fb_0.Error)));
	testState_0 := testState_0 + 1;
2:
	fb_0.Activate := TRUE; fb_0.S_Button1 := TRUE; fb_0.S_Button2 := FALSE;
	fb_0();
	failed_0 := NOT ((((((fb_0.DiagCode = 49168) AND fb_0.Ready) AND NOT (fb_0.S_TwoHandOut)) AND NOT (fb_0.SafetyDemand)) AND fb_0.Error));
	testState_0 := testState_0 + 1;
3:
	fb_0.Activate := TRUE; fb_0.S_Button1 := TRUE; fb_0.S_Button2 := FALSE;
	fb_0();
	failed_0 := NOT ((((((fb_0.DiagCode = 49168) AND fb_0.Ready) AND NOT (fb_0.S_TwoHandOut)) AND NOT (fb_0.SafetyDemand)) AND fb_0.Error));
	testState_0 := testState_0 + 1;
4:
	fb_0.Activate := TRUE; fb_0.S_Button1 := FALSE; fb_0.S_Button2 := FALSE;
	fb_0();
	failed_0 := NOT ((((((fb_0.DiagCode = 34818) AND fb_0.Ready) AND NOT (fb_0.S_TwoHandOut)) AND fb_0.SafetyDemand) AND NOT (fb_0.Error)));
	testState_0 := testState_0 + 1;
5:
	fb_0.Activate := FALSE;
	fb_0();
	failed_0 := NOT ((((((fb_0.DiagCode = 0) AND NOT (fb_0.Ready)) AND NOT (fb_0.S_TwoHandOut)) AND NOT (fb_0.SafetyDemand)) AND NOT (fb_0.Error)));
	testState_0 := testState_0 + 1;
6:
	fb_0.Activate := TRUE; fb_0.S_Button1 := FALSE; fb_0.S_Button2 := FALSE;
	fb_0();
	failed_0 := NOT ((((((fb_0.DiagCode = 32769) AND fb_0.Ready) AND NOT (fb_0.S_TwoHandOut)) AND NOT (fb_0.SafetyDemand)) AND NOT (fb_0.Error)));
	testState_0 := testState_0 + 1;
7:
	fb_0.Activate := TRUE; fb_0.S_Button1 := FALSE; fb_0.S_Button2 := TRUE;
	fb_0();
	failed_0 := NOT ((((((fb_0.DiagCode = 49184) AND fb_0.Ready) AND NOT (fb_0.S_TwoHandOut)) AND NOT (fb_0.SafetyDemand)) AND fb_0.Error));
	testState_0 := testState_0 + 1;
8:
	fb_0.Activate := TRUE; fb_0.S_Button1 := FALSE; fb_0.S_Button2 := TRUE;
	fb_0();
	failed_0 := NOT ((((((fb_0.DiagCode = 49184) AND fb_0.Ready) AND NOT (fb_0.S_TwoHandOut)) AND NOT (fb_0.SafetyDemand)) AND fb_0.Error));
	testState_0 := testState_0 + 1;
9:
	fb_0.Activate := TRUE; fb_0.S_Button1 := FALSE; fb_0.S_Button2 := FALSE;
	fb_0();
	failed_0 := NOT ((((((fb_0.DiagCode = 34818) AND fb_0.Ready) AND NOT (fb_0.S_TwoHandOut)) AND fb_0.SafetyDemand) AND NOT (fb_0.Error)));
	testState_0 := testState_0 + 1;
10:
	fb_0.Activate := FALSE;
	fb_0();
	failed_0 := NOT ((((((fb_0.DiagCode = 0) AND NOT (fb_0.Ready)) AND NOT (fb_0.S_TwoHandOut)) AND NOT (fb_0.SafetyDemand)) AND NOT (fb_0.Error)));
	testState_0 := testState_0 + 1;
11:
	fb_0.Activate := TRUE; fb_0.S_Button1 := FALSE; fb_0.S_Button2 := FALSE;
	fb_0();
	failed_0 := NOT ((((((fb_0.DiagCode = 32769) AND fb_0.Ready) AND NOT (fb_0.S_TwoHandOut)) AND NOT (fb_0.SafetyDemand)) AND NOT (fb_0.Error)));
	testState_0 := testState_0 + 1;
12:
	fb_0.Activate := TRUE; fb_0.S_Button1 := TRUE; fb_0.S_Button2 := TRUE;
	fb_0();
	failed_0 := NOT ((((((fb_0.DiagCode = 49200) AND fb_0.Ready) AND NOT (fb_0.S_TwoHandOut)) AND NOT (fb_0.SafetyDemand)) AND fb_0.Error));
	testState_0 := testState_0 + 1;
13:
	fb_0.Activate := TRUE; fb_0.S_Button1 := TRUE; fb_0.S_Button2 := TRUE;
	fb_0();
	failed_0 := NOT ((((((fb_0.DiagCode = 49200) AND fb_0.Ready) AND NOT (fb_0.S_TwoHandOut)) AND NOT (fb_0.SafetyDemand)) AND fb_0.Error));
	testState_0 := testState_0 + 1;
14:
	fb_0.Activate := TRUE; fb_0.S_Button1 := FALSE; fb_0.S_Button2 := FALSE;
	fb_0();
	failed_0 := NOT ((((((fb_0.DiagCode = 34818) AND fb_0.Ready) AND NOT (fb_0.S_TwoHandOut)) AND fb_0.SafetyDemand) AND NOT (fb_0.Error)));
	testState_0 := testState_0 + 1;
15:
	fb_0.Activate := FALSE;
	fb_0();
	failed_0 := NOT ((((((fb_0.DiagCode = 0) AND NOT (fb_0.Ready)) AND NOT (fb_0.S_TwoHandOut)) AND NOT (fb_0.SafetyDemand)) AND NOT (fb_0.Error)));
	testState_0 := testState_0 + 1;
16:
	fb_0.Activate := TRUE; fb_0.S_Button1 := FALSE; fb_0.S_Button2 := FALSE;
	fb_0();
	failed_0 := NOT ((((((fb_0.DiagCode = 32769) AND fb_0.Ready) AND NOT (fb_0.S_TwoHandOut)) AND NOT (fb_0.SafetyDemand)) AND NOT (fb_0.Error)));
	testState_0 := testState_0 + 1;
17:
	fb_0.Activate := TRUE; fb_0.S_Button1 := FALSE; fb_0.S_Button2 := FALSE;
	fb_0();
	failed_0 := NOT ((((((fb_0.DiagCode = 34818) AND fb_0.Ready) AND NOT (fb_0.S_TwoHandOut)) AND fb_0.SafetyDemand) AND NOT (fb_0.Error)));
	testState_0 := testState_0 + 1;
18:
	fb_0.Activate := TRUE; fb_0.S_Button1 := FALSE; fb_0.S_Button2 := FALSE;
	fb_0();
	failed_0 := NOT ((((((fb_0.DiagCode = 34818) AND fb_0.Ready) AND NOT (fb_0.S_TwoHandOut)) AND fb_0.SafetyDemand) AND NOT (fb_0.Error)));
	testState_0 := testState_0 + 1;
19:
	fb_0.Activate := TRUE; fb_0.S_Button1 := TRUE; fb_0.S_Button2 := TRUE;
	fb_0();
	failed_0 := NOT ((((((fb_0.DiagCode = 32768) AND fb_0.Ready) AND fb_0.S_TwoHandOut) AND NOT (fb_0.SafetyDemand)) AND NOT (fb_0.Error)));
	testState_0 := testState_0 + 1;
20:
	fb_0.Activate := TRUE; fb_0.S_Button1 := TRUE; fb_0.S_Button2 := TRUE;
	fb_0();
	failed_0 := NOT ((((((fb_0.DiagCode = 32768) AND fb_0.Ready) AND fb_0.S_TwoHandOut) AND NOT (fb_0.SafetyDemand)) AND NOT (fb_0.Error)));
	testState_0 := testState_0 + 1;
21:
	fb_0.Activate := TRUE; fb_0.S_Button1 := TRUE; fb_0.S_Button2 := FALSE;
	fb_0();
	failed_0 := NOT ((((((fb_0.DiagCode = 34824) AND fb_0.Ready) AND NOT (fb_0.S_TwoHandOut)) AND fb_0.SafetyDemand) AND NOT (fb_0.Error)));
	testState_0 := testState_0 + 1;
22:
	fb_0.Activate := TRUE; fb_0.S_Button1 := TRUE; fb_0.S_Button2 := FALSE;
	fb_0();
	failed_0 := NOT ((((((fb_0.DiagCode = 34824) AND fb_0.Ready) AND NOT (fb_0.S_TwoHandOut)) AND fb_0.SafetyDemand) AND NOT (fb_0.Error)));
	testState_0 := testState_0 + 1;
23:
	fb_0.Activate := TRUE; fb_0.S_Button1 := TRUE; fb_0.S_Button2 := TRUE;
	fb_0();
	failed_0 := NOT ((((((fb_0.DiagCode = 34828) AND fb_0.Ready) AND NOT (fb_0.S_TwoHandOut)) AND fb_0.SafetyDemand) AND NOT (fb_0.Error)));
	testState_0 := testState_0 + 1;
24:
	fb_0.Activate := TRUE; fb_0.S_Button1 := TRUE; fb_0.S_Button2 := TRUE;
	fb_0();
	failed_0 := NOT ((((((fb_0.DiagCode = 34828) AND fb_0.Ready) AND NOT (fb_0.S_TwoHandOut)) AND fb_0.SafetyDemand) AND NOT (fb_0.Error)));
	testState_0 := testState_0 + 1;
25:
	fb_0.Activate := TRUE; fb_0.S_Button1 := FALSE; fb_0.S_Button2 := TRUE;
	fb_0();
	failed_0 := NOT ((((((fb_0.DiagCode = 34826) AND fb_0.Ready) AND NOT (fb_0.S_TwoHandOut)) AND fb_0.SafetyDemand) AND NOT (fb_0.Error)));
	testState_0 := testState_0 + 1;
26:
	fb_0.Activate := TRUE; fb_0.S_Button1 := FALSE; fb_0.S_Button2 := TRUE;
	fb_0();
	failed_0 := NOT ((((((fb_0.DiagCode = 34826) AND fb_0.Ready) AND NOT (fb_0.S_TwoHandOut)) AND fb_0.SafetyDemand) AND NOT (fb_0.Error)));
	testState_0 := testState_0 + 1;
27:
	fb_0.Activate := TRUE; fb_0.S_Button1 := TRUE; fb_0.S_Button2 := TRUE;
	fb_0();
	failed_0 := NOT ((((((fb_0.DiagCode = 34828) AND fb_0.Ready) AND NOT (fb_0.S_TwoHandOut)) AND fb_0.SafetyDemand) AND NOT (fb_0.Error)));
	testState_0 := testState_0 + 1;
28:
	fb_0.Activate := TRUE; fb_0.S_Button1 := TRUE; fb_0.S_Button2 := FALSE;
	fb_0();
	failed_0 := NOT ((((((fb_0.DiagCode = 34824) AND fb_0.Ready) AND NOT (fb_0.S_TwoHandOut)) AND fb_0.SafetyDemand) AND NOT (fb_0.Error)));
	testState_0 := testState_0 + 1;
29:
	fb_0.Activate := TRUE; fb_0.S_Button1 := FALSE; fb_0.S_Button2 := TRUE;
	fb_0();
	failed_0 := NOT ((((((fb_0.DiagCode = 34826) AND fb_0.Ready) AND NOT (fb_0.S_TwoHandOut)) AND fb_0.SafetyDemand) AND NOT (fb_0.Error)));
	testState_0 := testState_0 + 1;
30:
	fb_0.Activate := TRUE; fb_0.S_Button1 := TRUE; fb_0.S_Button2 := FALSE;
	fb_0();
	failed_0 := NOT ((((((fb_0.DiagCode = 34824) AND fb_0.Ready) AND NOT (fb_0.S_TwoHandOut)) AND fb_0.SafetyDemand) AND NOT (fb_0.Error)));
	testState_0 := testState_0 + 1;
31:
	fb_0.Activate := TRUE; fb_0.S_Button1 := FALSE; fb_0.S_Button2 := FALSE;
	fb_0();
	failed_0 := NOT ((((((fb_0.DiagCode = 34818) AND fb_0.Ready) AND NOT (fb_0.S_TwoHandOut)) AND fb_0.SafetyDemand) AND NOT (fb_0.Error)));
	testState_0 := testState_0 + 1;
32:
	fb_0.Activate := TRUE; fb_0.S_Button1 := TRUE; fb_0.S_Button2 := TRUE;
	fb_0();
	failed_0 := NOT ((((((fb_0.DiagCode = 32768) AND fb_0.Ready) AND fb_0.S_TwoHandOut) AND NOT (fb_0.SafetyDemand)) AND NOT (fb_0.Error)));
	testState_0 := testState_0 + 1;
33:
	fb_0.Activate := TRUE; fb_0.S_Button1 := FALSE; fb_0.S_Button2 := TRUE;
	fb_0();
	failed_0 := NOT ((((((fb_0.DiagCode = 34826) AND fb_0.Ready) AND NOT (fb_0.S_TwoHandOut)) AND fb_0.SafetyDemand) AND NOT (fb_0.Error)));
	testState_0 := testState_0 + 1;
34:
	fb_0.Activate := TRUE; fb_0.S_Button1 := FALSE; fb_0.S_Button2 := FALSE;
	fb_0();
	failed_0 := NOT ((((((fb_0.DiagCode = 34818) AND fb_0.Ready) AND NOT (fb_0.S_TwoHandOut)) AND fb_0.SafetyDemand) AND NOT (fb_0.Error)));
	testState_0 := testState_0 + 1;
35:
	fb_0.Activate := TRUE; fb_0.S_Button1 := TRUE; fb_0.S_Button2 := TRUE;
	fb_0();
	failed_0 := NOT ((((((fb_0.DiagCode = 32768) AND fb_0.Ready) AND fb_0.S_TwoHandOut) AND NOT (fb_0.SafetyDemand)) AND NOT (fb_0.Error)));
	testState_0 := testState_0 + 1;
36:
	fb_0.Activate := TRUE; fb_0.S_Button1 := TRUE; fb_0.S_Button2 := FALSE;
	fb_0();
	failed_0 := NOT ((((((fb_0.DiagCode = 34824) AND fb_0.Ready) AND NOT (fb_0.S_TwoHandOut)) AND fb_0.SafetyDemand) AND NOT (fb_0.Error)));
	testState_0 := testState_0 + 1;
37:
	fb_0.Activate := TRUE; fb_0.S_Button1 := TRUE; fb_0.S_Button2 := TRUE;
	fb_0();
	failed_0 := NOT ((((((fb_0.DiagCode = 34828) AND fb_0.Ready) AND NOT (fb_0.S_TwoHandOut)) AND fb_0.SafetyDemand) AND NOT (fb_0.Error)));
	testState_0 := testState_0 + 1;
38:
	fb_0.Activate := TRUE; fb_0.S_Button1 := FALSE; fb_0.S_Button2 := FALSE;
	fb_0();
	failed_0 := NOT ((((((fb_0.DiagCode = 34818) AND fb_0.Ready) AND NOT (fb_0.S_TwoHandOut)) AND fb_0.SafetyDemand) AND NOT (fb_0.Error)));
	testState_0 := testState_0 + 1;
39:
	fb_0.Activate := TRUE; fb_0.S_Button1 := TRUE; fb_0.S_Button2 := TRUE;
	fb_0();
	failed_0 := NOT ((((((fb_0.DiagCode = 32768) AND fb_0.Ready) AND fb_0.S_TwoHandOut) AND NOT (fb_0.SafetyDemand)) AND NOT (fb_0.Error)));
	testState_0 := testState_0 + 1;
40:
	fb_0.Activate := TRUE; fb_0.S_Button1 := FALSE; fb_0.S_Button2 := FALSE;
	fb_0();
	failed_0 := NOT ((((((fb_0.DiagCode = 34818) AND fb_0.Ready) AND NOT (fb_0.S_TwoHandOut)) AND fb_0.SafetyDemand) AND NOT (fb_0.Error)));
	testState_0 := testState_0 + 1;
41:
	fb_0.Activate := TRUE; fb_0.S_Button1 := TRUE; fb_0.S_Button2 := FALSE;
	fb_0();
	failed_0 := NOT ((((((fb_0.DiagCode = 34820) AND fb_0.Ready) AND NOT (fb_0.S_TwoHandOut)) AND fb_0.SafetyDemand) AND NOT (fb_0.Error)));
	testState_0 := testState_0 + 1;
42:
	fb_0.Activate := TRUE; fb_0.S_Button1 := TRUE; fb_0.S_Button2 := FALSE;
	fb_0();
	failed_0 := NOT ((((((fb_0.DiagCode = 34820) AND fb_0.Ready) AND NOT (fb_0.S_TwoHandOut)) AND fb_0.SafetyDemand) AND NOT (fb_0.Error)));
	testState_0 := testState_0 + 1;
43:
	fb_0.Activate := TRUE; fb_0.S_Button1 := FALSE; fb_0.S_Button2 := FALSE;
	fb_0();
	failed_0 := NOT ((((((fb_0.DiagCode = 34818) AND fb_0.Ready) AND NOT (fb_0.S_TwoHandOut)) AND fb_0.SafetyDemand) AND NOT (fb_0.Error)));
	testState_0 := testState_0 + 1;
44:
	fb_0.Activate := TRUE; fb_0.S_Button1 := TRUE; fb_0.S_Button2 := FALSE;
	fb_0();
	failed_0 := NOT ((((((fb_0.DiagCode = 34820) AND fb_0.Ready) AND NOT (fb_0.S_TwoHandOut)) AND fb_0.SafetyDemand) AND NOT (fb_0.Error)));
	testState_0 := testState_0 + 1;
45:
	fb_0.Activate := TRUE; fb_0.S_Button1 := FALSE; fb_0.S_Button2 := TRUE;
	fb_0();
	failed_0 := NOT ((((((fb_0.DiagCode = 34830) AND fb_0.Ready) AND NOT (fb_0.S_TwoHandOut)) AND fb_0.SafetyDemand) AND NOT (fb_0.Error)));
	testState_0 := testState_0 + 1;
46:
	fb_0.Activate := TRUE; fb_0.S_Button1 := FALSE; fb_0.S_Button2 := TRUE;
	fb_0();
	failed_0 := NOT ((((((fb_0.DiagCode = 34830) AND fb_0.Ready) AND NOT (fb_0.S_TwoHandOut)) AND fb_0.SafetyDemand) AND NOT (fb_0.Error)));
	testState_0 := testState_0 + 1;
47:
	fb_0.Activate := TRUE; fb_0.S_Button1 := FALSE; fb_0.S_Button2 := FALSE;
	fb_0();
	failed_0 := NOT ((((((fb_0.DiagCode = 34818) AND fb_0.Ready) AND NOT (fb_0.S_TwoHandOut)) AND fb_0.SafetyDemand) AND NOT (fb_0.Error)));
	testState_0 := testState_0 + 1;
48:
	fb_0.Activate := TRUE; fb_0.S_Button1 := TRUE; fb_0.S_Button2 := FALSE;
	fb_0();
	failed_0 := NOT ((((((fb_0.DiagCode = 34820) AND fb_0.Ready) AND NOT (fb_0.S_TwoHandOut)) AND fb_0.SafetyDemand) AND NOT (fb_0.Error)));
	testState_0 := testState_0 + 1;
49:
	fb_0.Activate := TRUE; fb_0.S_Button1 := TRUE; fb_0.S_Button2 := TRUE;
	fb_0();
	failed_0 := NOT ((((((fb_0.DiagCode = 32768) AND fb_0.Ready) AND fb_0.S_TwoHandOut) AND NOT (fb_0.SafetyDemand)) AND NOT (fb_0.Error)));
	testState_0 := testState_0 + 1;
50:
	fb_0.Activate := TRUE; fb_0.S_Button1 := FALSE; fb_0.S_Button2 := FALSE;
	fb_0();
	failed_0 := NOT ((((((fb_0.DiagCode = 34818) AND fb_0.Ready) AND NOT (fb_0.S_TwoHandOut)) AND fb_0.SafetyDemand) AND NOT (fb_0.Error)));
	testState_0 := testState_0 + 1;
51:
	fb_0.Activate := TRUE; fb_0.S_Button1 := FALSE; fb_0.S_Button2 := TRUE;
	fb_0();
	failed_0 := NOT ((((((fb_0.DiagCode = 34822) AND fb_0.Ready) AND NOT (fb_0.S_TwoHandOut)) AND fb_0.SafetyDemand) AND NOT (fb_0.Error)));
	testState_0 := testState_0 + 1;
52:
	fb_0.Activate := TRUE; fb_0.S_Button1 := FALSE; fb_0.S_Button2 := TRUE;
	fb_0();
	failed_0 := NOT ((((((fb_0.DiagCode = 34822) AND fb_0.Ready) AND NOT (fb_0.S_TwoHandOut)) AND fb_0.SafetyDemand) AND NOT (fb_0.Error)));
	testState_0 := testState_0 + 1;
53:
	fb_0.Activate := TRUE; fb_0.S_Button1 := FALSE; fb_0.S_Button2 := FALSE;
	fb_0();
	failed_0 := NOT ((((((fb_0.DiagCode = 34818) AND fb_0.Ready) AND NOT (fb_0.S_TwoHandOut)) AND fb_0.SafetyDemand) AND NOT (fb_0.Error)));
	testState_0 := testState_0 + 1;
54:
	fb_0.Activate := TRUE; fb_0.S_Button1 := FALSE; fb_0.S_Button2 := TRUE;
	fb_0();
	failed_0 := NOT ((((((fb_0.DiagCode = 34822) AND fb_0.Ready) AND NOT (fb_0.S_TwoHandOut)) AND fb_0.SafetyDemand) AND NOT (fb_0.Error)));
	testState_0 := testState_0 + 1;
55:
	fb_0.Activate := TRUE; fb_0.S_Button1 := TRUE; fb_0.S_Button2 := FALSE;
	fb_0();
	failed_0 := NOT ((((((fb_0.DiagCode = 34830) AND fb_0.Ready) AND NOT (fb_0.S_TwoHandOut)) AND fb_0.SafetyDemand) AND NOT (fb_0.Error)));
	testState_0 := testState_0 + 1;
56:
	fb_0.Activate := TRUE; fb_0.S_Button1 := FALSE; fb_0.S_Button2 := FALSE;
	fb_0();
	failed_0 := NOT ((((((fb_0.DiagCode = 34818) AND fb_0.Ready) AND NOT (fb_0.S_TwoHandOut)) AND fb_0.SafetyDemand) AND NOT (fb_0.Error)));
	testState_0 := testState_0 + 1;
57:
	fb_0.Activate := TRUE; fb_0.S_Button1 := FALSE; fb_0.S_Button2 := TRUE;
	fb_0();
	failed_0 := NOT ((((((fb_0.DiagCode = 34822) AND fb_0.Ready) AND NOT (fb_0.S_TwoHandOut)) AND fb_0.SafetyDemand) AND NOT (fb_0.Error)));
	testState_0 := testState_0 + 1;
58:
	fb_0.Activate := TRUE; fb_0.S_Button1 := TRUE; fb_0.S_Button2 := TRUE;
	fb_0();
	failed_0 := NOT (((fb_0.DiagCode = 32768) AND (fb_0.Ready AND (fb_0.S_TwoHandOut AND (NOT (fb_0.SafetyDemand) AND NOT (fb_0.Error))))));
	testState_0 := testState_0 + 1;
59:
	finished_0 := TRUE;
END_CASE
END_IF

END_FUNCTION_BLOCK
